REGION Network 32: data management MV01
   RUNG wire#powerrail
      Contact( "EM_OK" )
      wire#w1
      I_Contact( "MV01_Close" )
      wire#w2
      Coil( "fill_unit1".CONTROL_SIGNALS.SW_GATE0 )
   END_RUNG
   RUNG wire#w2
      { S7_Templates := "SrcType := DInt"; S7_GenerateENO := "TRUE" } Add(in1 := "Memory encoder".Encoder_CH00, in2 := "fill_unit1".ACT_CNTV0, out => #CNT_Act_0)
      { S7_Templates := "SrcType := DInt"; S7_GenerateENO := "TRUE" } Div(in1 := #CNT_Act_0, in2 := 100, out => #CNTV0_100)
      { S7_GenerateENO := "TRUE" } Move(in := #CNTV0_100, out1 => "Memory encoder".Encoder_CH00_10)
   END_RUNG
   RUNG wire#w1
      I_Contact( "fill_unit1".CONTROL_SIGNALS.SW_GATE0 )
      wire#w3
      { S7_GenerateENO := "TRUE" } Move(in := 0, out1 => "Memory encoder".Encoder_CH00_10)
   END_RUNG
   RUNG wire#w3
      { S7_GenerateENO := "TRUE" } Move(in := INT#0, out1 => "Memory encoder".Encoder_CH00)
   END_RUNG
   RUNG wire#w1
      "Signal linearization"(IN0 := "ON", Analog_input := "Memory encoder".Encoder_CH00_10, Coeff := "Coeff".COEFF_TRASM_MV01, Zero := "Coeff".ZERO_TRASM_MV01, OutValue => "Data".Pot_MV01, Out_of_range => "Allarm".Pot_MV01_OFR)
   END_RUNG
   // the same network as SCL:
   // ENO of a box is taken as its EN; it also drops when the box reports an error
   "fill_unit1".CONTROL_SIGNALS.SW_GATE0 := "EM_OK" AND NOT "MV01_Close";
   IF "fill_unit1".CONTROL_SIGNALS.SW_GATE0 THEN
       #CNT_Act_0 := "Memory encoder".Encoder_CH00 + "fill_unit1".ACT_CNTV0;
       #CNTV0_100 := #CNT_Act_0 / 100;
       "Memory encoder".Encoder_CH00_10 := #CNTV0_100;
   END_IF;
   IF "EM_OK" AND NOT "fill_unit1".CONTROL_SIGNALS.SW_GATE0 THEN
       "Memory encoder".Encoder_CH00_10 := 0;
       "Memory encoder".Encoder_CH00 := INT#0;
   END_IF;
   IF "EM_OK" THEN
       "Signal linearization"(IN0 := "ON",
                              Analog_input := "Memory encoder".Encoder_CH00_10,
                              Coeff := "Coeff".COEFF_TRASM_MV01,
                              Zero := "Coeff".ZERO_TRASM_MV01,
                              OutValue => "Data".Pot_MV01,
                              Out_of_range => "Allarm".Pot_MV01_OFR);
   END_IF;
END_REGION

REGION Network 33: data management MV02
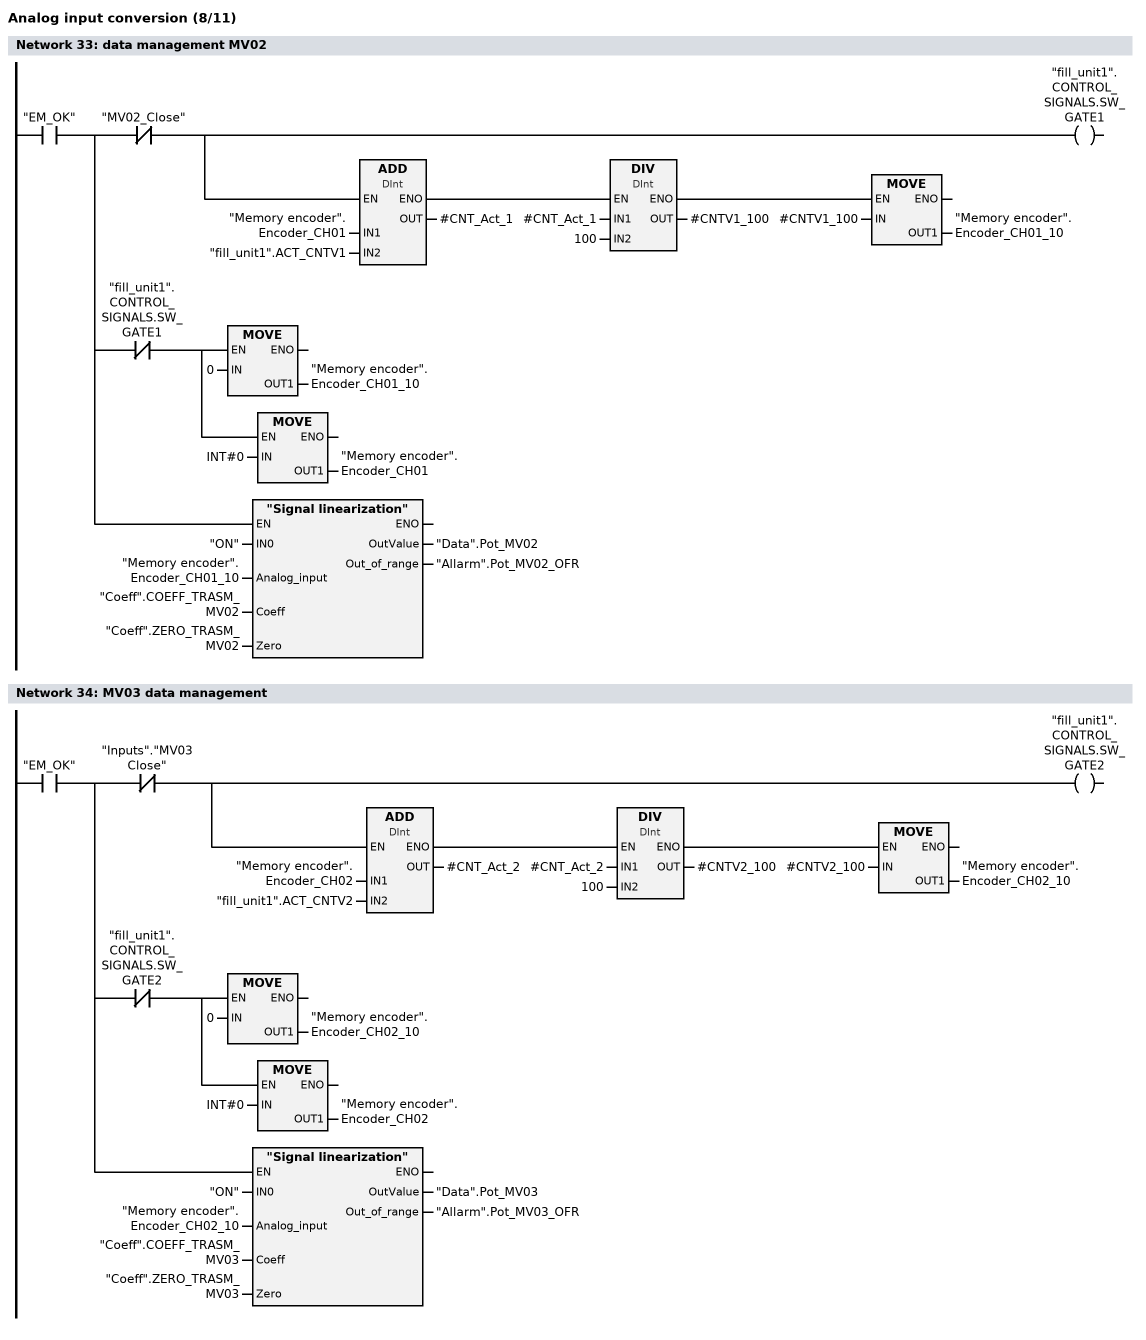
   RUNG wire#powerrail
      Contact( "EM_OK" )
      wire#w1
      I_Contact( "MV02_Close" )
      wire#w2
      Coil( "fill_unit1".CONTROL_SIGNALS.SW_GATE1 )
   END_RUNG
   RUNG wire#w2
      { S7_Templates := "SrcType := DInt"; S7_GenerateENO := "TRUE" } Add(in1 := "Memory encoder".Encoder_CH01, in2 := "fill_unit1".ACT_CNTV1, out => #CNT_Act_1)
      { S7_Templates := "SrcType := DInt"; S7_GenerateENO := "TRUE" } Div(in1 := #CNT_Act_1, in2 := 100, out => #CNTV1_100)
      { S7_GenerateENO := "TRUE" } Move(in := #CNTV1_100, out1 => "Memory encoder".Encoder_CH01_10)
   END_RUNG
   RUNG wire#w1
      I_Contact( "fill_unit1".CONTROL_SIGNALS.SW_GATE1 )
      wire#w3
      { S7_GenerateENO := "TRUE" } Move(in := 0, out1 => "Memory encoder".Encoder_CH01_10)
   END_RUNG
   RUNG wire#w3
      { S7_GenerateENO := "TRUE" } Move(in := INT#0, out1 => "Memory encoder".Encoder_CH01)
   END_RUNG
   RUNG wire#w1
      "Signal linearization"(IN0 := "ON", Analog_input := "Memory encoder".Encoder_CH01_10, Coeff := "Coeff".COEFF_TRASM_MV02, Zero := "Coeff".ZERO_TRASM_MV02, OutValue => "Data".Pot_MV02, Out_of_range => "Allarm".Pot_MV02_OFR)
   END_RUNG
   // the same network as SCL:
   // ENO of a box is taken as its EN; it also drops when the box reports an error
   "fill_unit1".CONTROL_SIGNALS.SW_GATE1 := "EM_OK" AND NOT "MV02_Close";
   IF "fill_unit1".CONTROL_SIGNALS.SW_GATE1 THEN
       #CNT_Act_1 := "Memory encoder".Encoder_CH01 + "fill_unit1".ACT_CNTV1;
       #CNTV1_100 := #CNT_Act_1 / 100;
       "Memory encoder".Encoder_CH01_10 := #CNTV1_100;
   END_IF;
   IF "EM_OK" AND NOT "fill_unit1".CONTROL_SIGNALS.SW_GATE1 THEN
       "Memory encoder".Encoder_CH01_10 := 0;
       "Memory encoder".Encoder_CH01 := INT#0;
   END_IF;
   IF "EM_OK" THEN
       "Signal linearization"(IN0 := "ON",
                              Analog_input := "Memory encoder".Encoder_CH01_10,
                              Coeff := "Coeff".COEFF_TRASM_MV02,
                              Zero := "Coeff".ZERO_TRASM_MV02,
                              OutValue => "Data".Pot_MV02,
                              Out_of_range => "Allarm".Pot_MV02_OFR);
   END_IF;
END_REGION

REGION Network 34: MV03 data management
   RUNG wire#powerrail
      Contact( "EM_OK" )
      wire#w1
      I_Contact( "Inputs"."MV03 Close" )
      wire#w2
      Coil( "fill_unit1".CONTROL_SIGNALS.SW_GATE2 )
   END_RUNG
   RUNG wire#w2
      { S7_Templates := "SrcType := DInt"; S7_GenerateENO := "TRUE" } Add(in1 := "Memory encoder".Encoder_CH02, in2 := "fill_unit1".ACT_CNTV2, out => #CNT_Act_2)
      { S7_Templates := "SrcType := DInt"; S7_GenerateENO := "TRUE" } Div(in1 := #CNT_Act_2, in2 := 100, out => #CNTV2_100)
      { S7_GenerateENO := "TRUE" } Move(in := #CNTV2_100, out1 => "Memory encoder".Encoder_CH02_10)
   END_RUNG
   RUNG wire#w1
      I_Contact( "fill_unit1".CONTROL_SIGNALS.SW_GATE2 )
      wire#w3
      { S7_GenerateENO := "TRUE" } Move(in := 0, out1 => "Memory encoder".Encoder_CH02_10)
   END_RUNG
   RUNG wire#w3
      { S7_GenerateENO := "TRUE" } Move(in := INT#0, out1 => "Memory encoder".Encoder_CH02)
   END_RUNG
   RUNG wire#w1
      "Signal linearization"(IN0 := "ON", Analog_input := "Memory encoder".Encoder_CH02_10, Coeff := "Coeff".COEFF_TRASM_MV03, Zero := "Coeff".ZERO_TRASM_MV03, OutValue => "Data".Pot_MV03, Out_of_range => "Allarm".Pot_MV03_OFR)
   END_RUNG
   // the same network as SCL:
   // ENO of a box is taken as its EN; it also drops when the box reports an error
   "fill_unit1".CONTROL_SIGNALS.SW_GATE2 := "EM_OK" AND NOT "Inputs"."MV03 Close";
   IF "fill_unit1".CONTROL_SIGNALS.SW_GATE2 THEN
       #CNT_Act_2 := "Memory encoder".Encoder_CH02 + "fill_unit1".ACT_CNTV2;
       #CNTV2_100 := #CNT_Act_2 / 100;
       "Memory encoder".Encoder_CH02_10 := #CNTV2_100;
   END_IF;
   IF "EM_OK" AND NOT "fill_unit1".CONTROL_SIGNALS.SW_GATE2 THEN
       "Memory encoder".Encoder_CH02_10 := 0;
       "Memory encoder".Encoder_CH02 := INT#0;
   END_IF;
   IF "EM_OK" THEN
       "Signal linearization"(IN0 := "ON",
                              Analog_input := "Memory encoder".Encoder_CH02_10,
                              Coeff := "Coeff".COEFF_TRASM_MV03,
                              Zero := "Coeff".ZERO_TRASM_MV03,
                              OutValue => "Data".Pot_MV03,
                              Out_of_range => "Allarm".Pot_MV03_OFR);
   END_IF;
END_REGION

REGION Network 35: MV05 data management
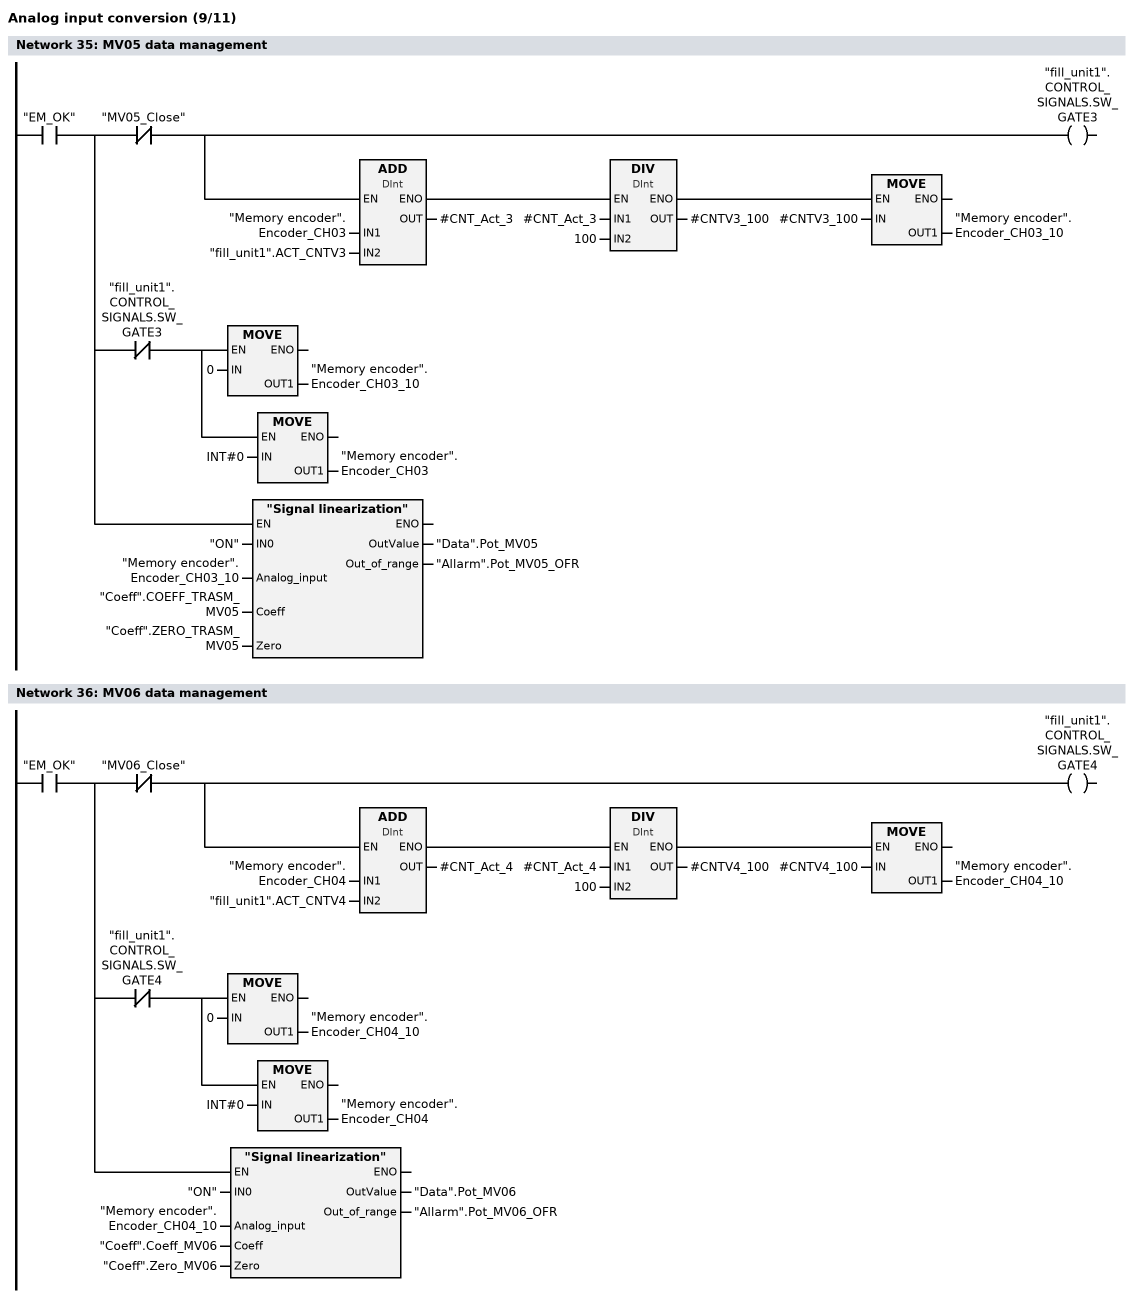
   RUNG wire#powerrail
      Contact( "EM_OK" )
      wire#w1
      I_Contact( "MV05_Close" )
      wire#w2
      Coil( "fill_unit1".CONTROL_SIGNALS.SW_GATE3 )
   END_RUNG
   RUNG wire#w2
      { S7_Templates := "SrcType := DInt"; S7_GenerateENO := "TRUE" } Add(in1 := "Memory encoder".Encoder_CH03, in2 := "fill_unit1".ACT_CNTV3, out => #CNT_Act_3)
      { S7_Templates := "SrcType := DInt"; S7_GenerateENO := "TRUE" } Div(in1 := #CNT_Act_3, in2 := 100, out => #CNTV3_100)
      { S7_GenerateENO := "TRUE" } Move(in := #CNTV3_100, out1 => "Memory encoder".Encoder_CH03_10)
   END_RUNG
   RUNG wire#w1
      I_Contact( "fill_unit1".CONTROL_SIGNALS.SW_GATE3 )
      wire#w3
      { S7_GenerateENO := "TRUE" } Move(in := 0, out1 => "Memory encoder".Encoder_CH03_10)
   END_RUNG
   RUNG wire#w3
      { S7_GenerateENO := "TRUE" } Move(in := INT#0, out1 => "Memory encoder".Encoder_CH03)
   END_RUNG
   RUNG wire#w1
      "Signal linearization"(IN0 := "ON", Analog_input := "Memory encoder".Encoder_CH03_10, Coeff := "Coeff".COEFF_TRASM_MV05, Zero := "Coeff".ZERO_TRASM_MV05, OutValue => "Data".Pot_MV05, Out_of_range => "Allarm".Pot_MV05_OFR)
   END_RUNG
   // the same network as SCL:
   // ENO of a box is taken as its EN; it also drops when the box reports an error
   "fill_unit1".CONTROL_SIGNALS.SW_GATE3 := "EM_OK" AND NOT "MV05_Close";
   IF "fill_unit1".CONTROL_SIGNALS.SW_GATE3 THEN
       #CNT_Act_3 := "Memory encoder".Encoder_CH03 + "fill_unit1".ACT_CNTV3;
       #CNTV3_100 := #CNT_Act_3 / 100;
       "Memory encoder".Encoder_CH03_10 := #CNTV3_100;
   END_IF;
   IF "EM_OK" AND NOT "fill_unit1".CONTROL_SIGNALS.SW_GATE3 THEN
       "Memory encoder".Encoder_CH03_10 := 0;
       "Memory encoder".Encoder_CH03 := INT#0;
   END_IF;
   IF "EM_OK" THEN
       "Signal linearization"(IN0 := "ON",
                              Analog_input := "Memory encoder".Encoder_CH03_10,
                              Coeff := "Coeff".COEFF_TRASM_MV05,
                              Zero := "Coeff".ZERO_TRASM_MV05,
                              OutValue => "Data".Pot_MV05,
                              Out_of_range => "Allarm".Pot_MV05_OFR);
   END_IF;
END_REGION

REGION Network 36: MV06 data management
   RUNG wire#powerrail
      Contact( "EM_OK" )
      wire#w1
      I_Contact( "MV06_Close" )
      wire#w2
      Coil( "fill_unit1".CONTROL_SIGNALS.SW_GATE4 )
   END_RUNG
   RUNG wire#w2
      { S7_Templates := "SrcType := DInt"; S7_GenerateENO := "TRUE" } Add(in1 := "Memory encoder".Encoder_CH04, in2 := "fill_unit1".ACT_CNTV4, out => #CNT_Act_4)
      { S7_Templates := "SrcType := DInt"; S7_GenerateENO := "TRUE" } Div(in1 := #CNT_Act_4, in2 := 100, out => #CNTV4_100)
      { S7_GenerateENO := "TRUE" } Move(in := #CNTV4_100, out1 => "Memory encoder".Encoder_CH04_10)
   END_RUNG
   RUNG wire#w1
      I_Contact( "fill_unit1".CONTROL_SIGNALS.SW_GATE4 )
      wire#w3
      { S7_GenerateENO := "TRUE" } Move(in := 0, out1 => "Memory encoder".Encoder_CH04_10)
   END_RUNG
   RUNG wire#w3
      { S7_GenerateENO := "TRUE" } Move(in := INT#0, out1 => "Memory encoder".Encoder_CH04)
   END_RUNG
   RUNG wire#w1
      "Signal linearization"(IN0 := "ON", Analog_input := "Memory encoder".Encoder_CH04_10, Coeff := "Coeff".Coeff_MV06, Zero := "Coeff".Zero_MV06, OutValue => "Data".Pot_MV06, Out_of_range => "Allarm".Pot_MV06_OFR)
   END_RUNG
   // the same network as SCL:
   // ENO of a box is taken as its EN; it also drops when the box reports an error
   "fill_unit1".CONTROL_SIGNALS.SW_GATE4 := "EM_OK" AND NOT "MV06_Close";
   IF "fill_unit1".CONTROL_SIGNALS.SW_GATE4 THEN
       #CNT_Act_4 := "Memory encoder".Encoder_CH04 + "fill_unit1".ACT_CNTV4;
       #CNTV4_100 := #CNT_Act_4 / 100;
       "Memory encoder".Encoder_CH04_10 := #CNTV4_100;
   END_IF;
   IF "EM_OK" AND NOT "fill_unit1".CONTROL_SIGNALS.SW_GATE4 THEN
       "Memory encoder".Encoder_CH04_10 := 0;
       "Memory encoder".Encoder_CH04 := INT#0;
   END_IF;
   IF "EM_OK" THEN
       "Signal linearization"(IN0 := "ON",
                              Analog_input := "Memory encoder".Encoder_CH04_10,
                              Coeff := "Coeff".Coeff_MV06,
                              Zero := "Coeff".Zero_MV06,
                              OutValue => "Data".Pot_MV06,
                              Out_of_range => "Allarm".Pot_MV06_OFR);
   END_IF;
END_REGION

REGION Network 37: FN-02 FAN
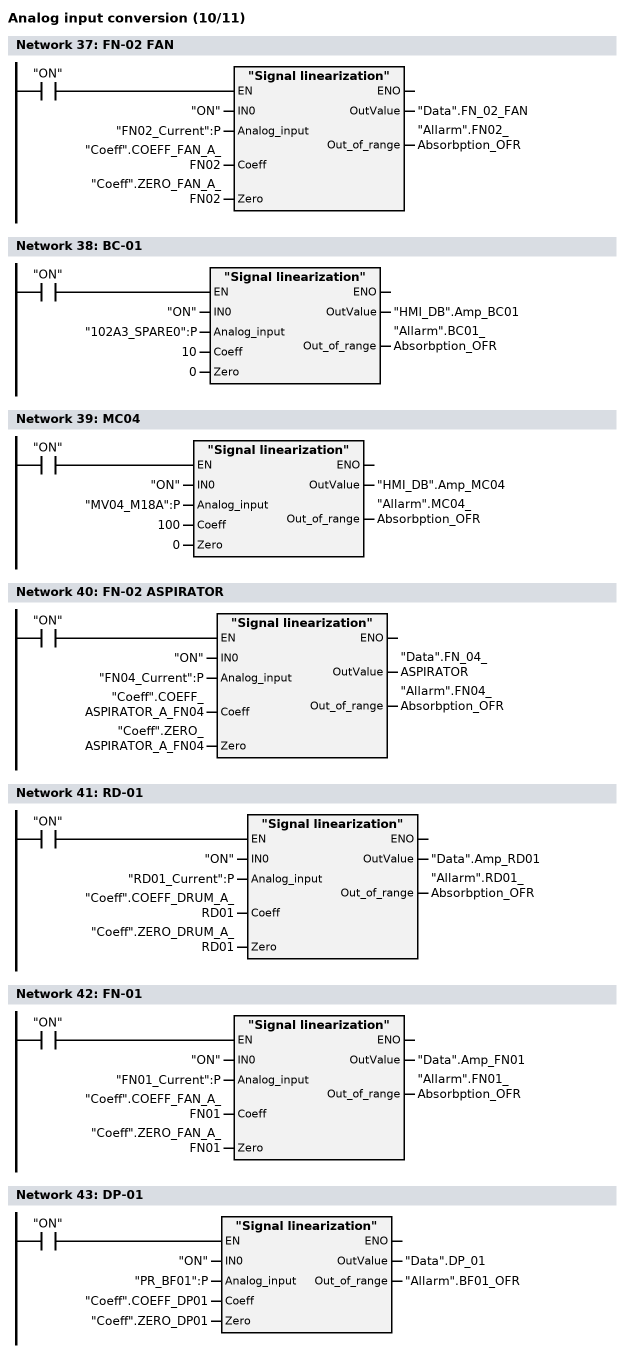
   RUNG wire#powerrail
      Contact( "ON" )
      "Signal linearization"(IN0 := "ON", Analog_input := "FN02_Current":P, Coeff := "Coeff".COEFF_FAN_A_FN02, Zero := "Coeff".ZERO_FAN_A_FN02, OutValue => "Data".FN_02_FAN, Out_of_range => "Allarm".FN02_Absorbption_OFR)
   END_RUNG
   // the same network as SCL:
   IF "ON" THEN
       "Signal linearization"(IN0 := "ON",
                              Analog_input := "FN02_Current":P,
                              Coeff := "Coeff".COEFF_FAN_A_FN02,
                              Zero := "Coeff".ZERO_FAN_A_FN02,
                              OutValue => "Data".FN_02_FAN,
                              Out_of_range => "Allarm".FN02_Absorbption_OFR);
   END_IF;
END_REGION

REGION Network 38: BC-01
   RUNG wire#powerrail
      Contact( "ON" )
      "Signal linearization"(IN0 := "ON", Analog_input := "102A3_SPARE0":P, Coeff := 10, Zero := 0, OutValue => "HMI_DB".Amp_BC01, Out_of_range => "Allarm".BC01_Absorbption_OFR)
   END_RUNG
   // the same network as SCL:
   IF "ON" THEN
       "Signal linearization"(IN0 := "ON",
                              Analog_input := "102A3_SPARE0":P,
                              Coeff := 10,
                              Zero := 0,
                              OutValue => "HMI_DB".Amp_BC01,
                              Out_of_range => "Allarm".BC01_Absorbption_OFR);
   END_IF;
END_REGION

REGION Network 39: MC04
   RUNG wire#powerrail
      Contact( "ON" )
      "Signal linearization"(IN0 := "ON", Analog_input := "MV04_M18A":P, Coeff := 100, Zero := 0, OutValue => "HMI_DB".Amp_MC04, Out_of_range => "Allarm".MC04_Absorbption_OFR)
   END_RUNG
   // the same network as SCL:
   IF "ON" THEN
       "Signal linearization"(IN0 := "ON",
                              Analog_input := "MV04_M18A":P,
                              Coeff := 100,
                              Zero := 0,
                              OutValue => "HMI_DB".Amp_MC04,
                              Out_of_range => "Allarm".MC04_Absorbption_OFR);
   END_IF;
END_REGION

REGION Network 40: FN-02 ASPIRATOR
   RUNG wire#powerrail
      Contact( "ON" )
      "Signal linearization"(IN0 := "ON", Analog_input := "FN04_Current":P, Coeff := "Coeff".COEFF_ASPIRATOR_A_FN04, Zero := "Coeff".ZERO_ASPIRATOR_A_FN04, OutValue => "Data".FN_04_ASPIRATOR, Out_of_range => "Allarm".FN04_Absorbption_OFR)
   END_RUNG
   // the same network as SCL:
   IF "ON" THEN
       "Signal linearization"(IN0 := "ON",
                              Analog_input := "FN04_Current":P,
                              Coeff := "Coeff".COEFF_ASPIRATOR_A_FN04,
                              Zero := "Coeff".ZERO_ASPIRATOR_A_FN04,
                              OutValue => "Data".FN_04_ASPIRATOR,
                              Out_of_range => "Allarm".FN04_Absorbption_OFR);
   END_IF;
END_REGION

REGION Network 41: RD-01
   RUNG wire#powerrail
      Contact( "ON" )
      "Signal linearization"(IN0 := "ON", Analog_input := "RD01_Current":P, Coeff := "Coeff".COEFF_DRUM_A_RD01, Zero := "Coeff".ZERO_DRUM_A_RD01, OutValue => "Data".Amp_RD01, Out_of_range => "Allarm".RD01_Absorbption_OFR)
   END_RUNG
   // the same network as SCL:
   IF "ON" THEN
       "Signal linearization"(IN0 := "ON",
                              Analog_input := "RD01_Current":P,
                              Coeff := "Coeff".COEFF_DRUM_A_RD01,
                              Zero := "Coeff".ZERO_DRUM_A_RD01,
                              OutValue => "Data".Amp_RD01,
                              Out_of_range => "Allarm".RD01_Absorbption_OFR);
   END_IF;
END_REGION

REGION Network 42: FN-01
   RUNG wire#powerrail
      Contact( "ON" )
      "Signal linearization"(IN0 := "ON", Analog_input := "FN01_Current":P, Coeff := "Coeff".COEFF_FAN_A_FN01, Zero := "Coeff".ZERO_FAN_A_FN01, OutValue => "Data".Amp_FN01, Out_of_range => "Allarm".FN01_Absorbption_OFR)
   END_RUNG
   // the same network as SCL:
   IF "ON" THEN
       "Signal linearization"(IN0 := "ON",
                              Analog_input := "FN01_Current":P,
                              Coeff := "Coeff".COEFF_FAN_A_FN01,
                              Zero := "Coeff".ZERO_FAN_A_FN01,
                              OutValue => "Data".Amp_FN01,
                              Out_of_range => "Allarm".FN01_Absorbption_OFR);
   END_IF;
END_REGION

REGION Network 43: DP-01
   RUNG wire#powerrail
      Contact( "ON" )
      "Signal linearization"(IN0 := "ON", Analog_input := "PR_BF01":P, Coeff := "Coeff".COEFF_DP01, Zero := "Coeff".ZERO_DP01, OutValue => "Data".DP_01, Out_of_range => "Allarm".BF01_OFR)
   END_RUNG
   // the same network as SCL:
   IF "ON" THEN
       "Signal linearization"(IN0 := "ON",
                              Analog_input := "PR_BF01":P,
                              Coeff := "Coeff".COEFF_DP01,
                              Zero := "Coeff".ZERO_DP01,
                              OutValue => "Data".DP_01,
                              Out_of_range => "Allarm".BF01_OFR);
   END_IF;
END_REGION

REGION Network 44: DP-02
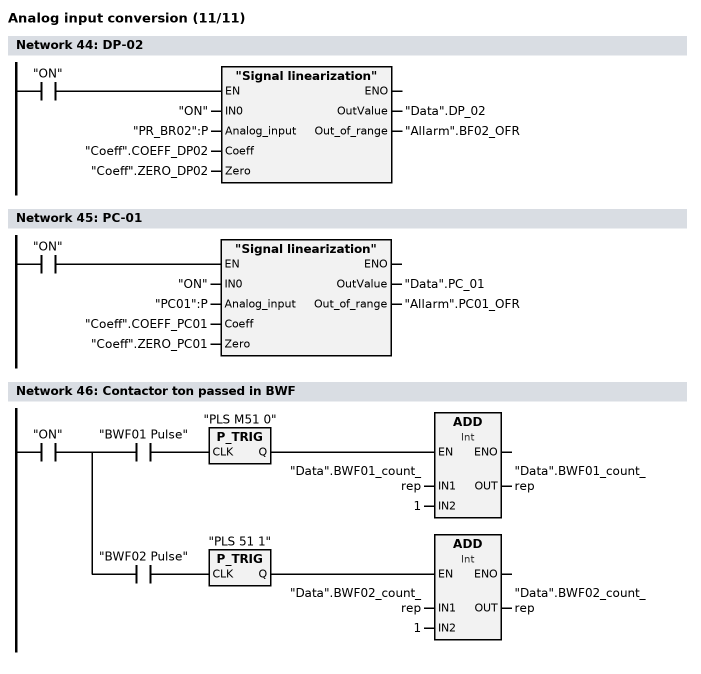
   RUNG wire#powerrail
      Contact( "ON" )
      "Signal linearization"(IN0 := "ON", Analog_input := "PR_BR02":P, Coeff := "Coeff".COEFF_DP02, Zero := "Coeff".ZERO_DP02, OutValue => "Data".DP_02, Out_of_range => "Allarm".BF02_OFR)
   END_RUNG
   // the same network as SCL:
   IF "ON" THEN
       "Signal linearization"(IN0 := "ON",
                              Analog_input := "PR_BR02":P,
                              Coeff := "Coeff".COEFF_DP02,
                              Zero := "Coeff".ZERO_DP02,
                              OutValue => "Data".DP_02,
                              Out_of_range => "Allarm".BF02_OFR);
   END_IF;
END_REGION

REGION Network 45: PC-01
   RUNG wire#powerrail
      Contact( "ON" )
      "Signal linearization"(IN0 := "ON", Analog_input := "PC01":P, Coeff := "Coeff".COEFF_PC01, Zero := "Coeff".ZERO_PC01, OutValue => "Data".PC_01, Out_of_range => "Allarm".PC01_OFR)
   END_RUNG
   // the same network as SCL:
   IF "ON" THEN
       "Signal linearization"(IN0 := "ON",
                              Analog_input := "PC01":P,
                              Coeff := "Coeff".COEFF_PC01,
                              Zero := "Coeff".ZERO_PC01,
                              OutValue => "Data".PC_01,
                              Out_of_range => "Allarm".PC01_OFR);
   END_IF;
END_REGION

REGION Network 46: Contactor ton passed in BWF
   RUNG wire#powerrail
      Contact( "ON" )
      wire#w1
      Contact( "BWF01 Pulse" )
      P_Trig( "PLS M51 0" )
      { S7_Templates := "SrcType := Int"; S7_GenerateENO := "TRUE" } Add(in1 := "Data".BWF01_count_rep, in2 := 1, out => "Data".BWF01_count_rep)
   END_RUNG
   RUNG wire#w1
      Contact( "BWF02 Pulse" )
      P_Trig( "PLS 51 1" )
      { S7_Templates := "SrcType := Int"; S7_GenerateENO := "TRUE" } Add(in1 := "Data".BWF02_count_rep, in2 := 1, out => "Data".BWF02_count_rep)
   END_RUNG
   // the same network as SCL:
   #_w1 := "ON" AND "BWF01 Pulse";
   #_w2 := #_w1 AND NOT "PLS M51 0";   // rising edge
   "PLS M51 0" := #_w1;
   IF #_w2 THEN "Data".BWF01_count_rep := "Data".BWF01_count_rep + 1; END_IF;
   #_w3 := "ON" AND "BWF02 Pulse";
   #_w4 := #_w3 AND NOT "PLS 51 1";   // rising edge
   "PLS 51 1" := #_w3;
   IF #_w4 THEN "Data".BWF02_count_rep := "Data".BWF02_count_rep + 1; END_IF;
END_REGION
END_FUNCTION

FUNCTION "Allarms 1" : Void   // FC4, LAD
TITLE = Motors alarms
{ S7_Optimized_Access := 'FALSE' }
VERSION : 0.1
   VAR_TEMP   // added for the SCL form of the ladder/FBD networks
      _w1 : Bool;
      _w2 : Bool;
      _w3 : Bool;
      _w4 : Bool;
      _w5 : Bool;
   END_VAR
BEGIN

REGION Network 1: BWF01
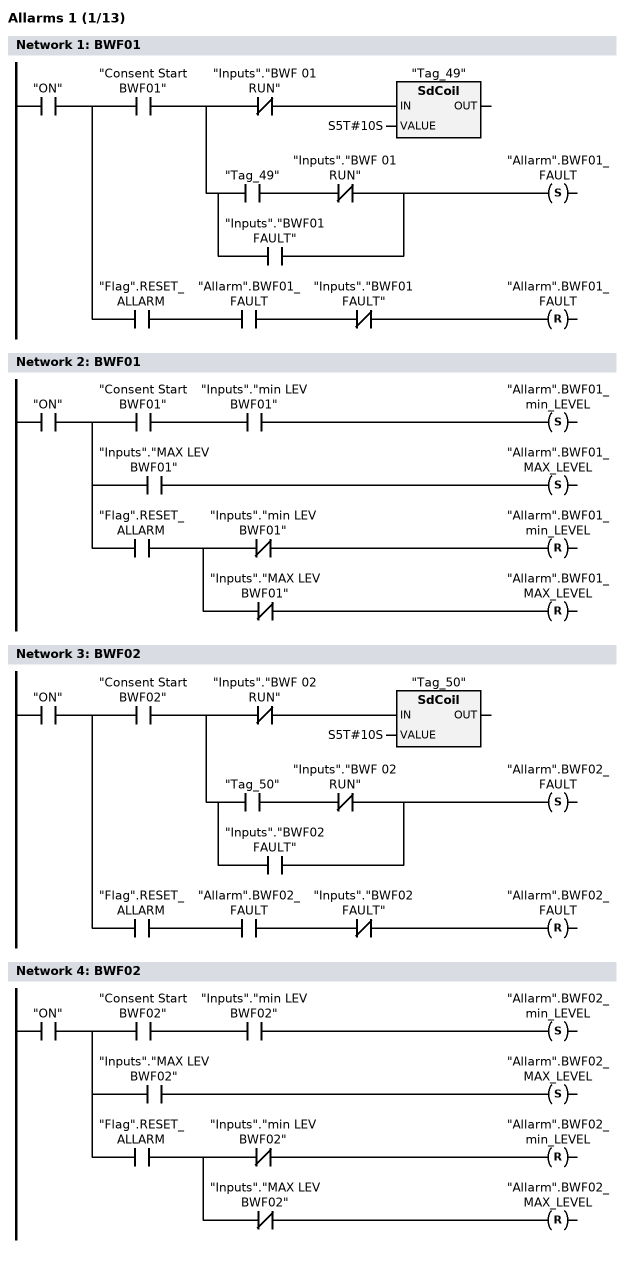
   // no SCL statement known for SdCoil: written as a call
   #_w1 := "ON" AND "Consent Start BWF01";
   #_w2 := "ON";
   SdCoil(in := #_w1 AND NOT "Inputs"."BWF 01 RUN", value := S5T#10S, operand := "Tag_49");
   IF #_w1 AND (("Tag_49" AND NOT "Inputs"."BWF 01 RUN") OR "Inputs"."BWF01 FAULT") THEN
       "Allarm".BWF01_FAULT := TRUE;
   END_IF;
   IF #_w2 AND "Flag".RESET_ALLARM AND "Allarm".BWF01_FAULT AND NOT "Inputs"."BWF01 FAULT" THEN
       "Allarm".BWF01_FAULT := FALSE;
   END_IF;
END_REGION

REGION Network 2: BWF01
   RUNG wire#powerrail
      Contact( "ON" )
      wire#w1
      Contact( "Consent Start BWF01" )
      Contact( "Inputs"."min LEV BWF01" )
      S_Coil( "Allarm".BWF01_min_LEVEL )
   END_RUNG
   RUNG wire#w1
      Contact( "Inputs"."MAX LEV BWF01" )
      S_Coil( "Allarm".BWF01_MAX_LEVEL )
   END_RUNG
   RUNG wire#w1
      Contact( "Flag".RESET_ALLARM )
      wire#w2
      I_Contact( "Inputs"."min LEV BWF01" )
      R_Coil( "Allarm".BWF01_min_LEVEL )
   END_RUNG
   RUNG wire#w2
      I_Contact( "Inputs"."MAX LEV BWF01" )
      R_Coil( "Allarm".BWF01_MAX_LEVEL )
   END_RUNG
   // the same network as SCL:
   IF "ON" AND "Consent Start BWF01" AND "Inputs"."min LEV BWF01" THEN
       "Allarm".BWF01_min_LEVEL := TRUE;
   END_IF;
   IF "ON" AND "Inputs"."MAX LEV BWF01" THEN "Allarm".BWF01_MAX_LEVEL := TRUE; END_IF;
   #_w1 := "ON" AND "Flag".RESET_ALLARM;
   IF #_w1 AND NOT "Inputs"."min LEV BWF01" THEN "Allarm".BWF01_min_LEVEL := FALSE; END_IF;
   IF #_w1 AND NOT "Inputs"."MAX LEV BWF01" THEN "Allarm".BWF01_MAX_LEVEL := FALSE; END_IF;
END_REGION

REGION Network 3: BWF02
   // no SCL statement known for SdCoil: written as a call
   #_w1 := "ON" AND "Consent Start BWF02";
   #_w2 := "ON";
   SdCoil(in := #_w1 AND NOT "Inputs"."BWF 02 RUN", value := S5T#10S, operand := "Tag_50");
   IF #_w1 AND (("Tag_50" AND NOT "Inputs"."BWF 02 RUN") OR "Inputs"."BWF02 FAULT") THEN
       "Allarm".BWF02_FAULT := TRUE;
   END_IF;
   IF #_w2 AND "Flag".RESET_ALLARM AND "Allarm".BWF02_FAULT AND NOT "Inputs"."BWF02 FAULT" THEN
       "Allarm".BWF02_FAULT := FALSE;
   END_IF;
END_REGION

REGION Network 4: BWF02
   RUNG wire#powerrail
      Contact( "ON" )
      wire#w1
      Contact( "Consent Start BWF02" )
      Contact( "Inputs"."min LEV BWF02" )
      S_Coil( "Allarm".BWF02_min_LEVEL )
   END_RUNG
   RUNG wire#w1
      Contact( "Inputs"."MAX LEV BWF02" )
      S_Coil( "Allarm".BWF02_MAX_LEVEL )
   END_RUNG
   RUNG wire#w1
      Contact( "Flag".RESET_ALLARM )
      wire#w2
      I_Contact( "Inputs"."min LEV BWF02" )
      R_Coil( "Allarm".BWF02_min_LEVEL )
   END_RUNG
   RUNG wire#w2
      I_Contact( "Inputs"."MAX LEV BWF02" )
      R_Coil( "Allarm".BWF02_MAX_LEVEL )
   END_RUNG
   // the same network as SCL:
   IF "ON" AND "Consent Start BWF02" AND "Inputs"."min LEV BWF02" THEN
       "Allarm".BWF02_min_LEVEL := TRUE;
   END_IF;
   IF "ON" AND "Inputs"."MAX LEV BWF02" THEN "Allarm".BWF02_MAX_LEVEL := TRUE; END_IF;
   #_w1 := "ON" AND "Flag".RESET_ALLARM;
   IF #_w1 AND NOT "Inputs"."min LEV BWF02" THEN "Allarm".BWF02_min_LEVEL := FALSE; END_IF;
   IF #_w1 AND NOT "Inputs"."MAX LEV BWF02" THEN "Allarm".BWF02_MAX_LEVEL := FALSE; END_IF;
END_REGION

REGION Network 5: BC01
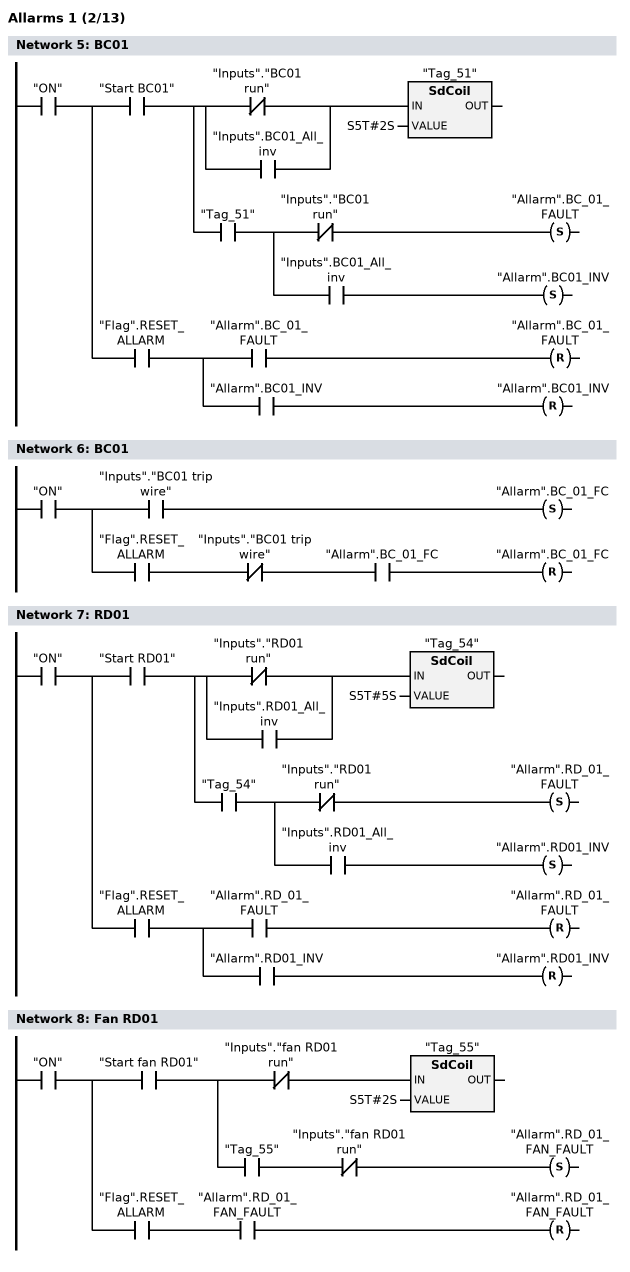
   // no SCL statement known for SdCoil: written as a call
   #_w1 := "ON" AND "Start BC01";
   #_w2 := "ON";
   SdCoil(in := #_w1 AND (NOT "Inputs"."BC01 run" OR "Inputs".BC01_All_inv),
          value := S5T#2S,
          operand := "Tag_51");
   #_w3 := #_w1 AND "Tag_51";
   IF #_w3 AND NOT "Inputs"."BC01 run" THEN "Allarm".BC_01_FAULT := TRUE; END_IF;
   IF #_w3 AND "Inputs".BC01_All_inv THEN "Allarm".BC01_INV := TRUE; END_IF;
   #_w4 := #_w2 AND "Flag".RESET_ALLARM;
   IF #_w4 AND "Allarm".BC_01_FAULT THEN "Allarm".BC_01_FAULT := FALSE; END_IF;
   IF #_w4 AND "Allarm".BC01_INV THEN "Allarm".BC01_INV := FALSE; END_IF;
END_REGION

REGION Network 6: BC01
   RUNG wire#powerrail
      Contact( "ON" )
      wire#w1
      Contact( "Inputs"."BC01 trip wire" )
      S_Coil( "Allarm".BC_01_FC )
   END_RUNG
   RUNG wire#w1
      Contact( "Flag".RESET_ALLARM )
      I_Contact( "Inputs"."BC01 trip wire" )
      Contact( "Allarm".BC_01_FC )
      R_Coil( "Allarm".BC_01_FC )
   END_RUNG
   // the same network as SCL:
   IF "ON" AND "Inputs"."BC01 trip wire" THEN "Allarm".BC_01_FC := TRUE; END_IF;
   IF "ON" AND "Flag".RESET_ALLARM AND NOT "Inputs"."BC01 trip wire" AND "Allarm".BC_01_FC THEN
       "Allarm".BC_01_FC := FALSE;
   END_IF;
END_REGION

REGION Network 7: RD01
   // no SCL statement known for SdCoil: written as a call
   #_w1 := "ON" AND "Start RD01";
   #_w2 := "ON";
   SdCoil(in := #_w1 AND (NOT "Inputs"."RD01 run" OR "Inputs".RD01_All_inv),
          value := S5T#5S,
          operand := "Tag_54");
   #_w3 := #_w1 AND "Tag_54";
   IF #_w3 AND NOT "Inputs"."RD01 run" THEN "Allarm".RD_01_FAULT := TRUE; END_IF;
   IF #_w3 AND "Inputs".RD01_All_inv THEN "Allarm".RD01_INV := TRUE; END_IF;
   #_w4 := #_w2 AND "Flag".RESET_ALLARM;
   IF #_w4 AND "Allarm".RD_01_FAULT THEN "Allarm".RD_01_FAULT := FALSE; END_IF;
   IF #_w4 AND "Allarm".RD01_INV THEN "Allarm".RD01_INV := FALSE; END_IF;
END_REGION

REGION Network 8: Fan RD01
   // no SCL statement known for SdCoil: written as a call
   #_w1 := "ON" AND "Start fan RD01";
   #_w2 := "ON";
   SdCoil(in := #_w1 AND NOT "Inputs"."fan RD01 run", value := S5T#2S, operand := "Tag_55");
   IF #_w1 AND "Tag_55" AND NOT "Inputs"."fan RD01 run" THEN "Allarm".RD_01_FAN_FAULT := TRUE; END_IF;
   IF #_w2 AND "Flag".RESET_ALLARM AND "Allarm".RD_01_FAN_FAULT THEN
       "Allarm".RD_01_FAN_FAULT := FALSE;
   END_IF;
END_REGION

REGION Network 9: Spare motor
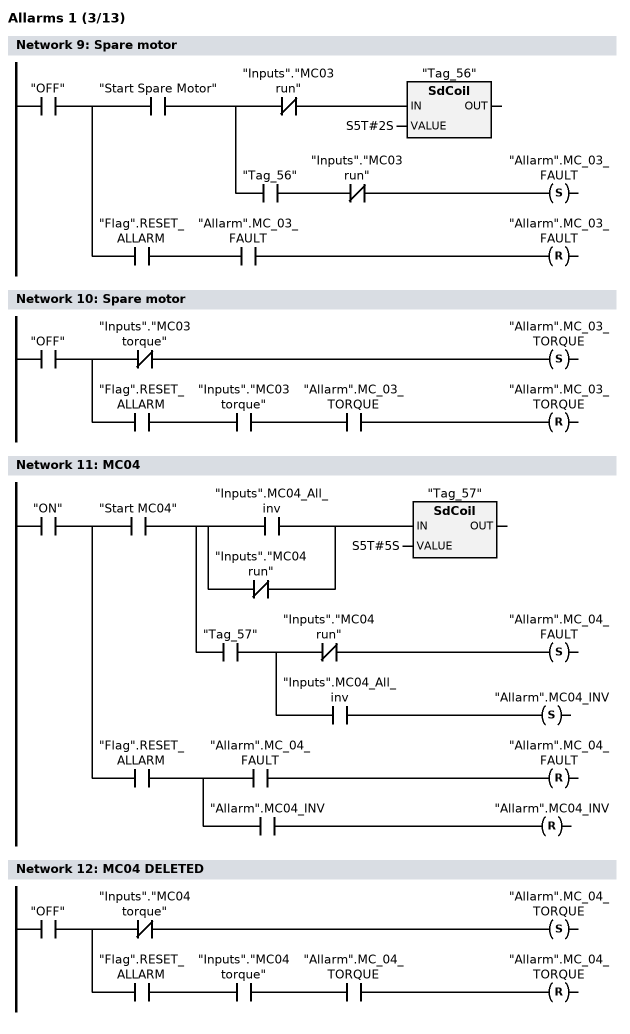
   // no SCL statement known for SdCoil: written as a call
   #_w1 := "OFF" AND "Start Spare Motor";
   #_w2 := "OFF";
   SdCoil(in := #_w1 AND NOT "Inputs"."MC03 run", value := S5T#2S, operand := "Tag_56");
   IF #_w1 AND "Tag_56" AND NOT "Inputs"."MC03 run" THEN "Allarm".MC_03_FAULT := TRUE; END_IF;
   IF #_w2 AND "Flag".RESET_ALLARM AND "Allarm".MC_03_FAULT THEN "Allarm".MC_03_FAULT := FALSE; END_IF;
END_REGION

REGION Network 10: Spare motor
   RUNG wire#powerrail
      Contact( "OFF" )
      wire#w1
      I_Contact( "Inputs"."MC03 torque" )
      S_Coil( "Allarm".MC_03_TORQUE )
   END_RUNG
   RUNG wire#w1
      Contact( "Flag".RESET_ALLARM )
      Contact( "Inputs"."MC03 torque" )
      Contact( "Allarm".MC_03_TORQUE )
      R_Coil( "Allarm".MC_03_TORQUE )
   END_RUNG
   // the same network as SCL:
   IF "OFF" AND NOT "Inputs"."MC03 torque" THEN "Allarm".MC_03_TORQUE := TRUE; END_IF;
   IF "OFF" AND "Flag".RESET_ALLARM AND "Inputs"."MC03 torque" AND "Allarm".MC_03_TORQUE THEN
       "Allarm".MC_03_TORQUE := FALSE;
   END_IF;
END_REGION

REGION Network 11: MC04
   // no SCL statement known for SdCoil: written as a call
   #_w1 := "ON" AND "Start MC04";
   #_w2 := "ON";
   SdCoil(in := #_w1 AND ("Inputs".MC04_All_inv OR NOT "Inputs"."MC04 run"),
          value := S5T#5S,
          operand := "Tag_57");
   #_w3 := #_w1 AND "Tag_57";
   IF #_w3 AND NOT "Inputs"."MC04 run" THEN "Allarm".MC_04_FAULT := TRUE; END_IF;
   IF #_w3 AND "Inputs".MC04_All_inv THEN "Allarm".MC04_INV := TRUE; END_IF;
   #_w4 := #_w2 AND "Flag".RESET_ALLARM;
   IF #_w4 AND "Allarm".MC_04_FAULT THEN "Allarm".MC_04_FAULT := FALSE; END_IF;
   IF #_w4 AND "Allarm".MC04_INV THEN "Allarm".MC04_INV := FALSE; END_IF;
END_REGION

REGION Network 12: MC04 DELETED
   RUNG wire#powerrail
      Contact( "OFF" )
      wire#w1
      I_Contact( "Inputs"."MC04 torque" )
      S_Coil( "Allarm".MC_04_TORQUE )
   END_RUNG
   RUNG wire#w1
      Contact( "Flag".RESET_ALLARM )
      Contact( "Inputs"."MC04 torque" )
      Contact( "Allarm".MC_04_TORQUE )
      R_Coil( "Allarm".MC_04_TORQUE )
   END_RUNG
   // the same network as SCL:
   IF "OFF" AND NOT "Inputs"."MC04 torque" THEN "Allarm".MC_04_TORQUE := TRUE; END_IF;
   IF "OFF" AND "Flag".RESET_ALLARM AND "Inputs"."MC04 torque" AND "Allarm".MC_04_TORQUE THEN
       "Allarm".MC_04_TORQUE := FALSE;
   END_IF;
END_REGION

REGION Network 13: MC05 DELETED
END_REGION

REGION Network 14: VS01
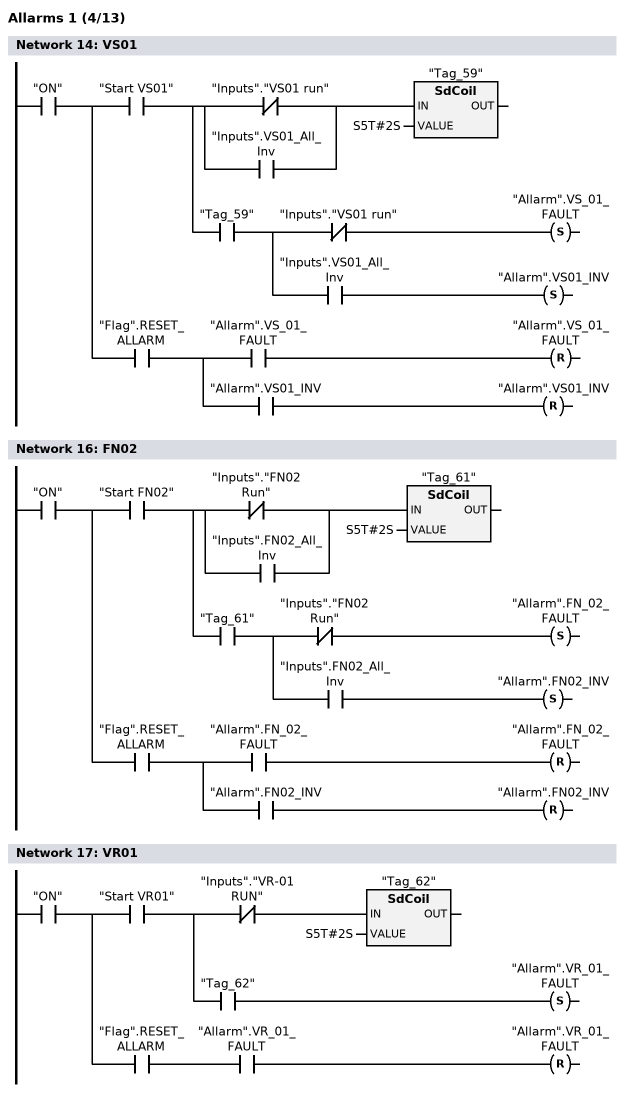
   // no SCL statement known for SdCoil: written as a call
   #_w1 := "ON" AND "Start VS01";
   #_w2 := "ON";
   SdCoil(in := #_w1 AND (NOT "Inputs"."VS01 run" OR "Inputs".VS01_All_Inv),
          value := S5T#2S,
          operand := "Tag_59");
   #_w3 := #_w1 AND "Tag_59";
   IF #_w3 AND NOT "Inputs"."VS01 run" THEN "Allarm".VS_01_FAULT := TRUE; END_IF;
   IF #_w3 AND "Inputs".VS01_All_Inv THEN "Allarm".VS01_INV := TRUE; END_IF;
   #_w4 := #_w2 AND "Flag".RESET_ALLARM;
   IF #_w4 AND "Allarm".VS_01_FAULT THEN "Allarm".VS_01_FAULT := FALSE; END_IF;
   IF #_w4 AND "Allarm".VS01_INV THEN "Allarm".VS01_INV := FALSE; END_IF;
END_REGION

REGION Network 15: SC12 DELETED
END_REGION

REGION Network 16: FN02
   // no SCL statement known for SdCoil: written as a call
   #_w1 := "ON" AND "Start FN02";
   #_w2 := "ON";
   SdCoil(in := #_w1 AND (NOT "Inputs"."FN02 Run" OR "Inputs".FN02_All_Inv),
          value := S5T#2S,
          operand := "Tag_61");
   #_w3 := #_w1 AND "Tag_61";
   IF #_w3 AND NOT "Inputs"."FN02 Run" THEN "Allarm".FN_02_FAULT := TRUE; END_IF;
   IF #_w3 AND "Inputs".FN02_All_Inv THEN "Allarm".FN02_INV := TRUE; END_IF;
   #_w4 := #_w2 AND "Flag".RESET_ALLARM;
   IF #_w4 AND "Allarm".FN_02_FAULT THEN "Allarm".FN_02_FAULT := FALSE; END_IF;
   IF #_w4 AND "Allarm".FN02_INV THEN "Allarm".FN02_INV := FALSE; END_IF;
END_REGION

REGION Network 17: VR01
   // no SCL statement known for SdCoil: written as a call
   #_w1 := "ON" AND "Start VR01";
   #_w2 := "ON";
   SdCoil(in := #_w1 AND NOT "Inputs"."VR-01 RUN", value := S5T#2S, operand := "Tag_62");
   IF #_w1 AND "Tag_62" THEN "Allarm".VR_01_FAULT := TRUE; END_IF;
   IF #_w2 AND "Flag".RESET_ALLARM AND "Allarm".VR_01_FAULT THEN "Allarm".VR_01_FAULT := FALSE; END_IF;
END_REGION

REGION Network 18: FN01
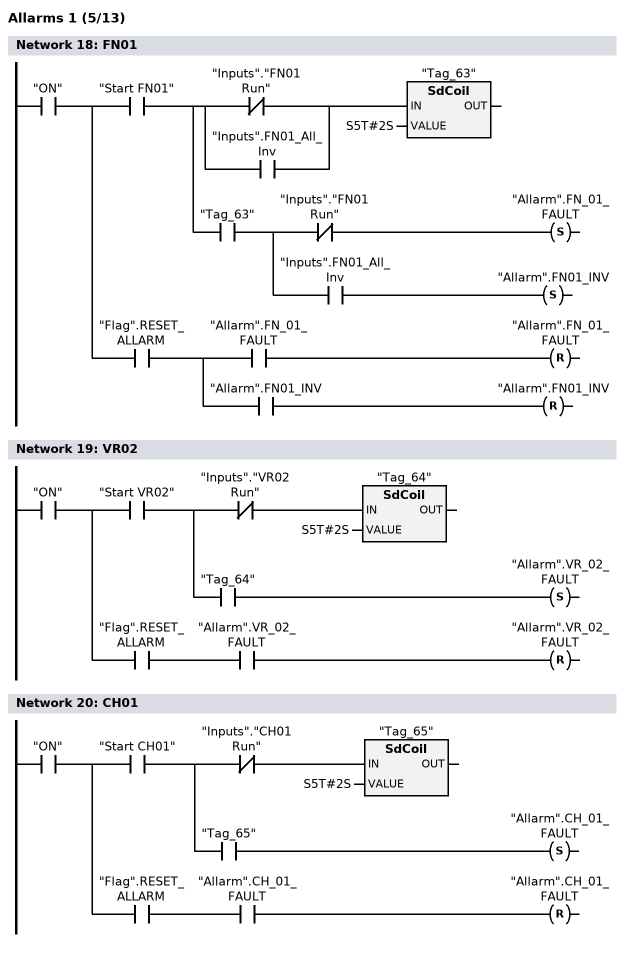
   // no SCL statement known for SdCoil: written as a call
   #_w1 := "ON" AND "Start FN01";
   #_w2 := "ON";
   SdCoil(in := #_w1 AND (NOT "Inputs"."FN01 Run" OR "Inputs".FN01_All_Inv),
          value := S5T#2S,
          operand := "Tag_63");
   #_w3 := #_w1 AND "Tag_63";
   IF #_w3 AND NOT "Inputs"."FN01 Run" THEN "Allarm".FN_01_FAULT := TRUE; END_IF;
   IF #_w3 AND "Inputs".FN01_All_Inv THEN "Allarm".FN01_INV := TRUE; END_IF;
   #_w4 := #_w2 AND "Flag".RESET_ALLARM;
   IF #_w4 AND "Allarm".FN_01_FAULT THEN "Allarm".FN_01_FAULT := FALSE; END_IF;
   IF #_w4 AND "Allarm".FN01_INV THEN "Allarm".FN01_INV := FALSE; END_IF;
END_REGION

REGION Network 19: VR02
   // no SCL statement known for SdCoil: written as a call
   #_w1 := "ON" AND "Start VR02";
   #_w2 := "ON";
   SdCoil(in := #_w1 AND NOT "Inputs"."VR02 Run", value := S5T#2S, operand := "Tag_64");
   IF #_w1 AND "Tag_64" THEN "Allarm".VR_02_FAULT := TRUE; END_IF;
   IF #_w2 AND "Flag".RESET_ALLARM AND "Allarm".VR_02_FAULT THEN "Allarm".VR_02_FAULT := FALSE; END_IF;
END_REGION

REGION Network 20: CH01
   // no SCL statement known for SdCoil: written as a call
   #_w1 := "ON" AND "Start CH01";
   #_w2 := "ON";
   SdCoil(in := #_w1 AND NOT "Inputs"."CH01 Run", value := S5T#2S, operand := "Tag_65");
   IF #_w1 AND "Tag_65" THEN "Allarm".CH_01_FAULT := TRUE; END_IF;
   IF #_w2 AND "Flag".RESET_ALLARM AND "Allarm".CH_01_FAULT THEN "Allarm".CH_01_FAULT := FALSE; END_IF;
END_REGION

REGION Network 21: FN03
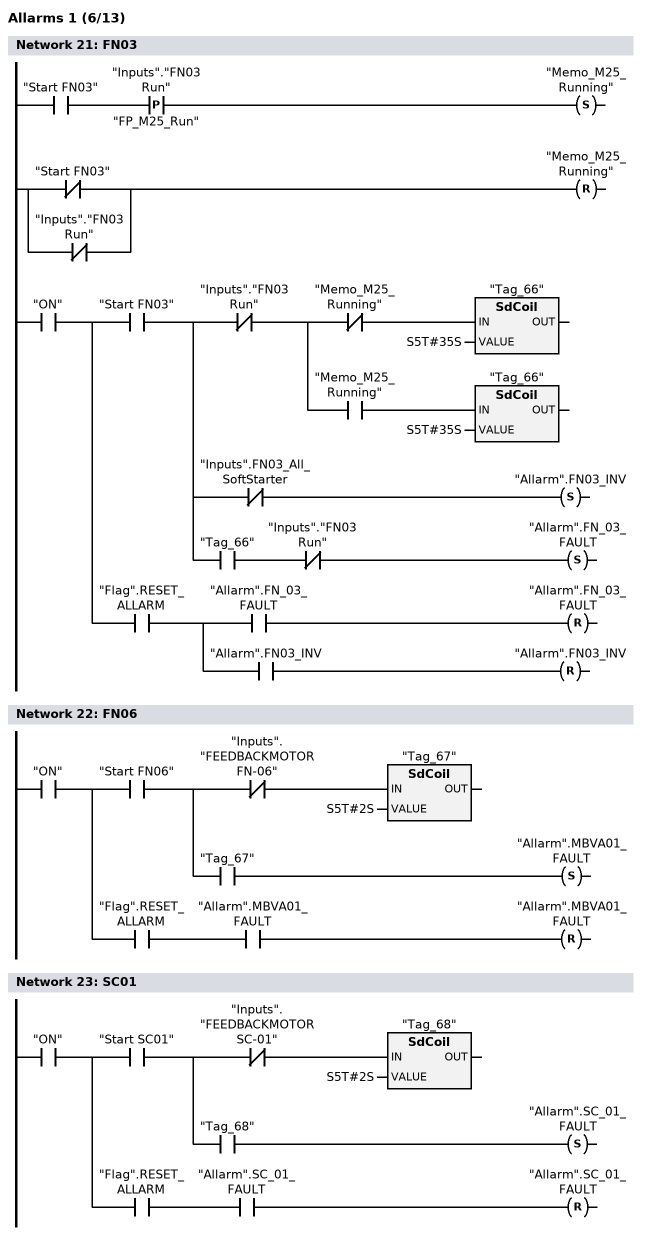
   // no SCL statement known for SdCoil: written as a call
   #_w1 := "Start FN03" AND "Inputs"."FN03 Run" AND NOT "FP_M25_Run";   // rising edge of "Inputs"."FN03 Run"
   "FP_M25_Run" := "Inputs"."FN03 Run";
   IF #_w1 THEN "Memo_M25_Running" := TRUE; END_IF;
   IF NOT "Start FN03" OR NOT "Inputs"."FN03 Run" THEN "Memo_M25_Running" := FALSE; END_IF;
   #_w2 := "ON" AND "Start FN03";
   #_w3 := #_w2 AND NOT "Inputs"."FN03 Run";
   #_w4 := "ON";
   SdCoil(in := #_w3 AND NOT "Memo_M25_Running", value := S5T#35S, operand := "Tag_66");
   SdCoil(in := #_w3 AND "Memo_M25_Running", value := S5T#35S, operand := "Tag_66");
   IF #_w2 AND NOT "Inputs".FN03_All_SoftStarter THEN "Allarm".FN03_INV := TRUE; END_IF;
   IF #_w2 AND "Tag_66" AND NOT "Inputs"."FN03 Run" THEN "Allarm".FN_03_FAULT := TRUE; END_IF;
   #_w5 := #_w4 AND "Flag".RESET_ALLARM;
   IF #_w5 AND "Allarm".FN_03_FAULT THEN "Allarm".FN_03_FAULT := FALSE; END_IF;
   IF #_w5 AND "Allarm".FN03_INV THEN "Allarm".FN03_INV := FALSE; END_IF;
END_REGION

REGION Network 22: FN06
   // no SCL statement known for SdCoil: written as a call
   #_w1 := "ON" AND "Start FN06";
   #_w2 := "ON";
   SdCoil(in := #_w1 AND NOT "Inputs"."FEEDBACKMOTOR FN-06", value := S5T#2S, operand := "Tag_67");
   IF #_w1 AND "Tag_67" THEN "Allarm".MBVA01_FAULT := TRUE; END_IF;
   IF #_w2 AND "Flag".RESET_ALLARM AND "Allarm".MBVA01_FAULT THEN "Allarm".MBVA01_FAULT := FALSE; END_IF;
END_REGION

REGION Network 23: SC01
   // no SCL statement known for SdCoil: written as a call
   #_w1 := "ON" AND "Start SC01";
   #_w2 := "ON";
   SdCoil(in := #_w1 AND NOT "Inputs"."FEEDBACKMOTOR SC-01", value := S5T#2S, operand := "Tag_68");
   IF #_w1 AND "Tag_68" THEN "Allarm".SC_01_FAULT := TRUE; END_IF;
   IF #_w2 AND "Flag".RESET_ALLARM AND "Allarm".SC_01_FAULT THEN "Allarm".SC_01_FAULT := FALSE; END_IF;
END_REGION

REGION Network 24: FN01_FAN DELETED
END_REGION

REGION Network 25: LD01
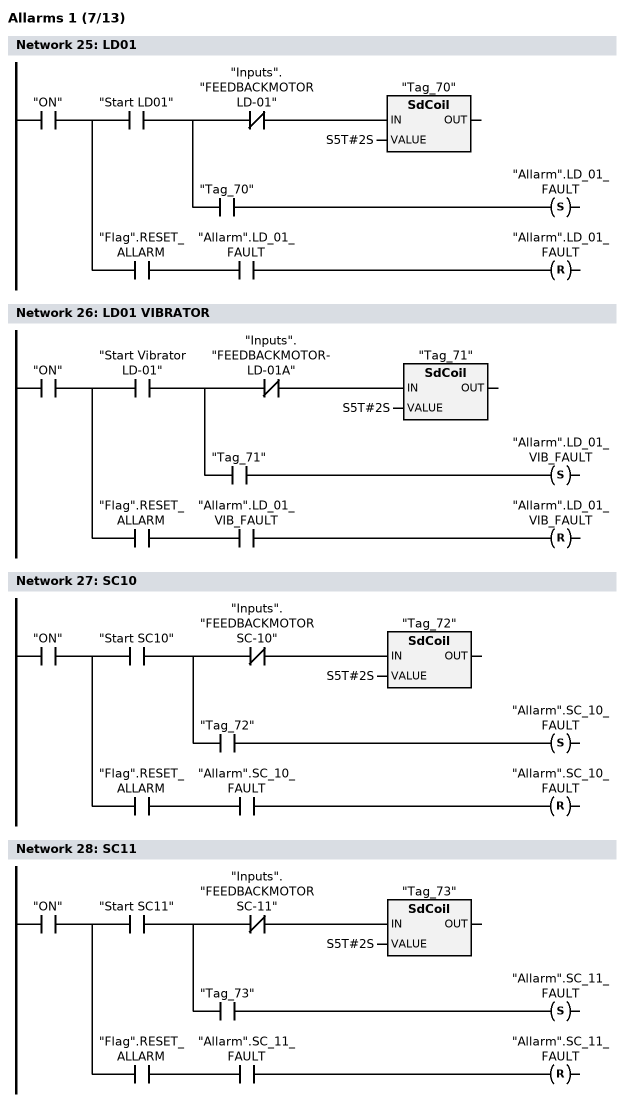
   // no SCL statement known for SdCoil: written as a call
   #_w1 := "ON" AND "Start LD01";
   #_w2 := "ON";
   SdCoil(in := #_w1 AND NOT "Inputs"."FEEDBACKMOTOR LD-01", value := S5T#2S, operand := "Tag_70");
   IF #_w1 AND "Tag_70" THEN "Allarm".LD_01_FAULT := TRUE; END_IF;
   IF #_w2 AND "Flag".RESET_ALLARM AND "Allarm".LD_01_FAULT THEN "Allarm".LD_01_FAULT := FALSE; END_IF;
END_REGION

REGION Network 26: LD01 VIBRATOR
   // no SCL statement known for SdCoil: written as a call
   #_w1 := "ON" AND "Start Vibrator LD-01";
   #_w2 := "ON";
   SdCoil(in := #_w1 AND NOT "Inputs"."FEEDBACKMOTOR-LD-01A", value := S5T#2S, operand := "Tag_71");
   IF #_w1 AND "Tag_71" THEN "Allarm".LD_01_VIB_FAULT := TRUE; END_IF;
   IF #_w2 AND "Flag".RESET_ALLARM AND "Allarm".LD_01_VIB_FAULT THEN
       "Allarm".LD_01_VIB_FAULT := FALSE;
   END_IF;
END_REGION

REGION Network 27: SC10
   // no SCL statement known for SdCoil: written as a call
   #_w1 := "ON" AND "Start SC10";
   #_w2 := "ON";
   SdCoil(in := #_w1 AND NOT "Inputs"."FEEDBACKMOTOR SC-10", value := S5T#2S, operand := "Tag_72");
   IF #_w1 AND "Tag_72" THEN "Allarm".SC_10_FAULT := TRUE; END_IF;
   IF #_w2 AND "Flag".RESET_ALLARM AND "Allarm".SC_10_FAULT THEN "Allarm".SC_10_FAULT := FALSE; END_IF;
END_REGION

REGION Network 28: SC11
   // no SCL statement known for SdCoil: written as a call
   #_w1 := "ON" AND "Start SC11";
   #_w2 := "ON";
   SdCoil(in := #_w1 AND NOT "Inputs"."FEEDBACKMOTOR SC-11", value := S5T#2S, operand := "Tag_73");
   IF #_w1 AND "Tag_73" THEN "Allarm".SC_11_FAULT := TRUE; END_IF;
   IF #_w2 AND "Flag".RESET_ALLARM AND "Allarm".SC_11_FAULT THEN "Allarm".SC_11_FAULT := FALSE; END_IF;
END_REGION

REGION Network 29: FN04
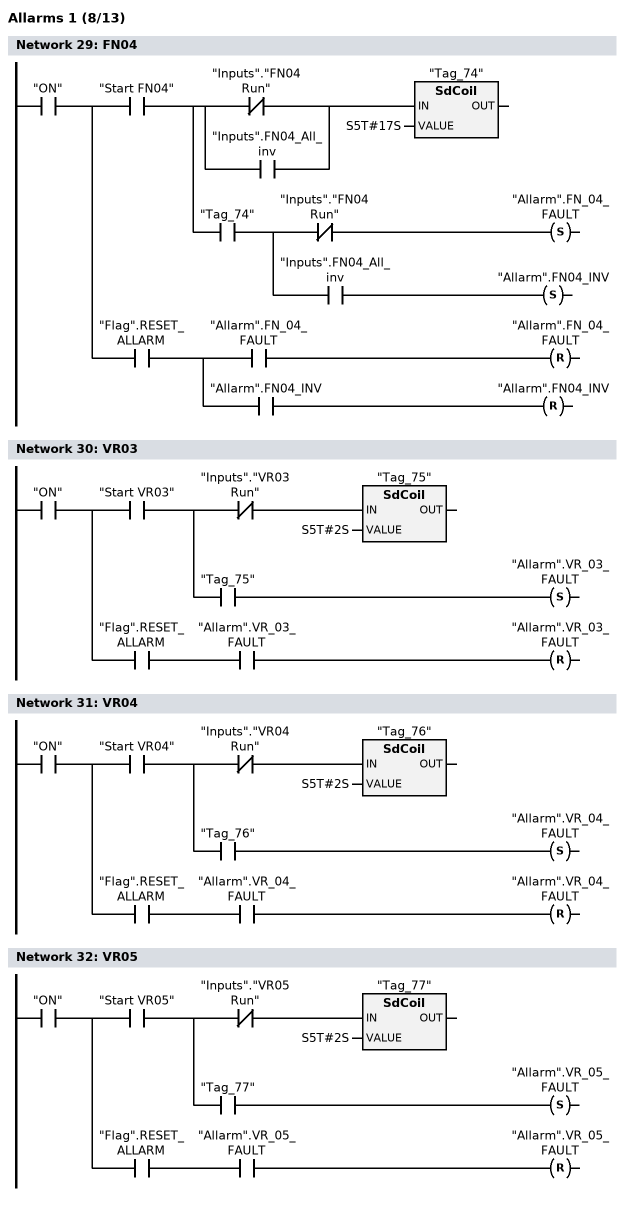
   // no SCL statement known for SdCoil: written as a call
   #_w1 := "ON" AND "Start FN04";
   #_w2 := "ON";
   SdCoil(in := #_w1 AND (NOT "Inputs"."FN04 Run" OR "Inputs".FN04_All_inv),
          value := S5T#17S,
          operand := "Tag_74");
   #_w3 := #_w1 AND "Tag_74";
   IF #_w3 AND NOT "Inputs"."FN04 Run" THEN "Allarm".FN_04_FAULT := TRUE; END_IF;
   IF #_w3 AND "Inputs".FN04_All_inv THEN "Allarm".FN04_INV := TRUE; END_IF;
   #_w4 := #_w2 AND "Flag".RESET_ALLARM;
   IF #_w4 AND "Allarm".FN_04_FAULT THEN "Allarm".FN_04_FAULT := FALSE; END_IF;
   IF #_w4 AND "Allarm".FN04_INV THEN "Allarm".FN04_INV := FALSE; END_IF;
END_REGION

REGION Network 30: VR03
   // no SCL statement known for SdCoil: written as a call
   #_w1 := "ON" AND "Start VR03";
   #_w2 := "ON";
   SdCoil(in := #_w1 AND NOT "Inputs"."VR03 Run", value := S5T#2S, operand := "Tag_75");
   IF #_w1 AND "Tag_75" THEN "Allarm".VR_03_FAULT := TRUE; END_IF;
   IF #_w2 AND "Flag".RESET_ALLARM AND "Allarm".VR_03_FAULT THEN "Allarm".VR_03_FAULT := FALSE; END_IF;
END_REGION

REGION Network 31: VR04
   // no SCL statement known for SdCoil: written as a call
   #_w1 := "ON" AND "Start VR04";
   #_w2 := "ON";
   SdCoil(in := #_w1 AND NOT "Inputs"."VR04 Run", value := S5T#2S, operand := "Tag_76");
   IF #_w1 AND "Tag_76" THEN "Allarm".VR_04_FAULT := TRUE; END_IF;
   IF #_w2 AND "Flag".RESET_ALLARM AND "Allarm".VR_04_FAULT THEN "Allarm".VR_04_FAULT := FALSE; END_IF;
END_REGION

REGION Network 32: VR05
   // no SCL statement known for SdCoil: written as a call
   #_w1 := "ON" AND "Start VR05";
   #_w2 := "ON";
   SdCoil(in := #_w1 AND NOT "Inputs"."VR05 Run", value := S5T#2S, operand := "Tag_77");
   IF #_w1 AND "Tag_77" THEN "Allarm".VR_05_FAULT := TRUE; END_IF;
   IF #_w2 AND "Flag".RESET_ALLARM AND "Allarm".VR_05_FAULT THEN "Allarm".VR_05_FAULT := FALSE; END_IF;
END_REGION

REGION Network 33: VR06
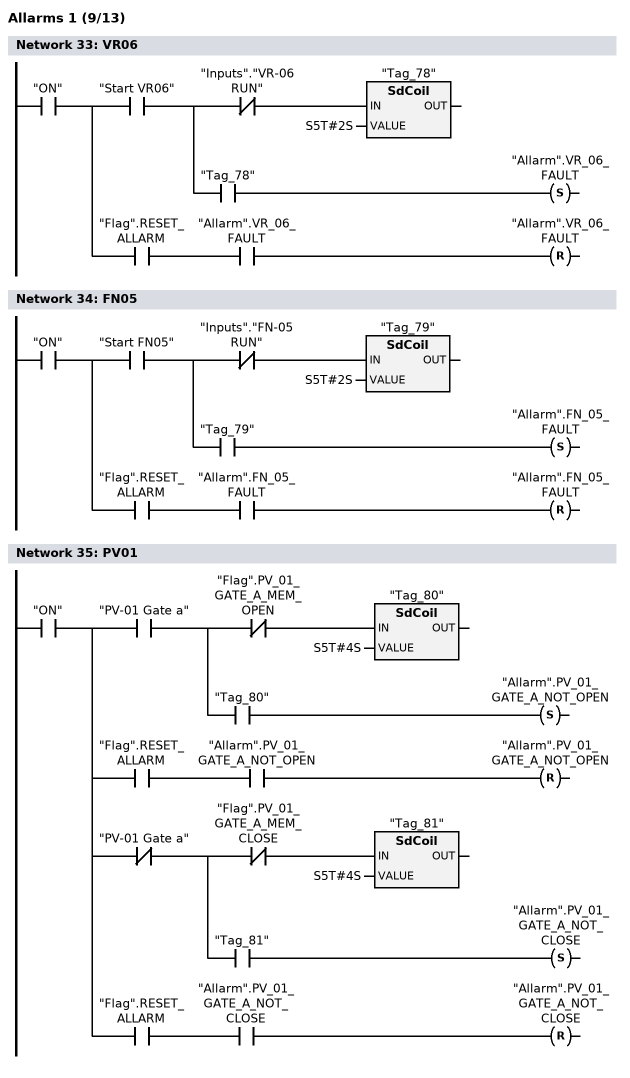
   // no SCL statement known for SdCoil: written as a call
   #_w1 := "ON" AND "Start VR06";
   #_w2 := "ON";
   SdCoil(in := #_w1 AND NOT "Inputs"."VR-06 RUN", value := S5T#2S, operand := "Tag_78");
   IF #_w1 AND "Tag_78" THEN "Allarm".VR_06_FAULT := TRUE; END_IF;
   IF #_w2 AND "Flag".RESET_ALLARM AND "Allarm".VR_06_FAULT THEN "Allarm".VR_06_FAULT := FALSE; END_IF;
END_REGION

REGION Network 34: FN05
   // no SCL statement known for SdCoil: written as a call
   #_w1 := "ON" AND "Start FN05";
   #_w2 := "ON";
   SdCoil(in := #_w1 AND NOT "Inputs"."FN-05 RUN", value := S5T#2S, operand := "Tag_79");
   IF #_w1 AND "Tag_79" THEN "Allarm".FN_05_FAULT := TRUE; END_IF;
   IF #_w2 AND "Flag".RESET_ALLARM AND "Allarm".FN_05_FAULT THEN "Allarm".FN_05_FAULT := FALSE; END_IF;
END_REGION

REGION Network 35: PV01
   // no SCL statement known for SdCoil: written as a call
   #_w1 := "ON" AND "PV-01 Gate a";
   #_w2 := "ON";
   SdCoil(in := #_w1 AND NOT "Flag".PV_01_GATE_A_MEM_OPEN, value := S5T#4S, operand := "Tag_80");
   IF #_w1 AND "Tag_80" THEN "Allarm".PV_01_GATE_A_NOT_OPEN := TRUE; END_IF;
   IF #_w2 AND "Flag".RESET_ALLARM AND "Allarm".PV_01_GATE_A_NOT_OPEN THEN
       "Allarm".PV_01_GATE_A_NOT_OPEN := FALSE;
   END_IF;
   #_w3 := #_w2 AND NOT "PV-01 Gate a";
   SdCoil(in := #_w3 AND NOT "Flag".PV_01_GATE_A_MEM_CLOSE, value := S5T#4S, operand := "Tag_81");
   IF #_w3 AND "Tag_81" THEN "Allarm".PV_01_GATE_A_NOT_CLOSE := TRUE; END_IF;
   IF #_w2 AND "Flag".RESET_ALLARM AND "Allarm".PV_01_GATE_A_NOT_CLOSE THEN
       "Allarm".PV_01_GATE_A_NOT_CLOSE := FALSE;
   END_IF;
END_REGION

REGION Network 36: PV01
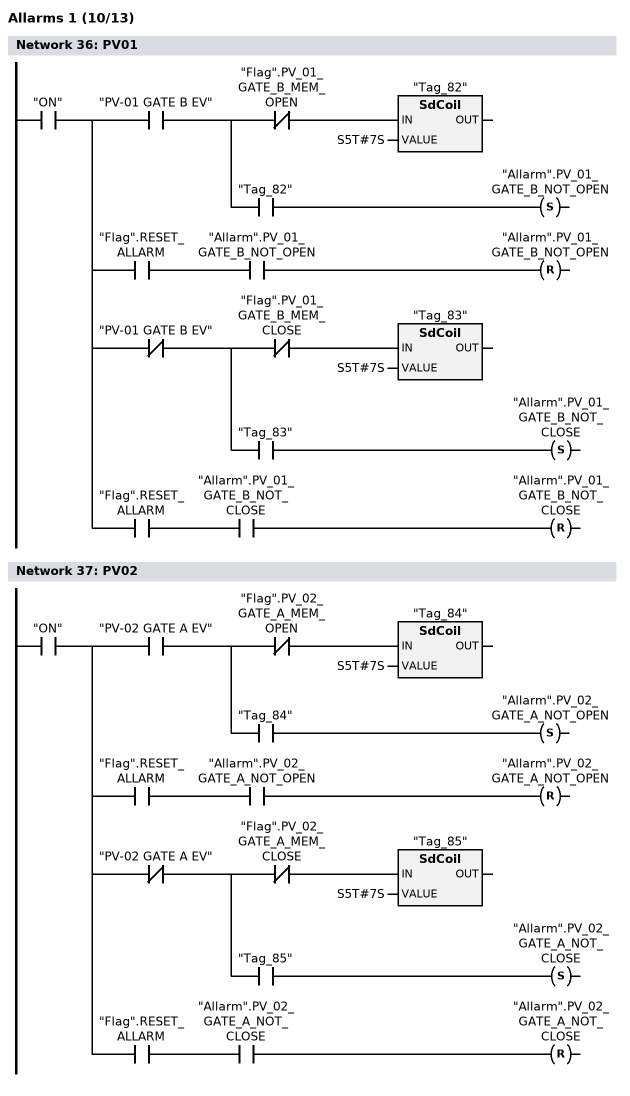
   // no SCL statement known for SdCoil: written as a call
   #_w1 := "ON" AND "PV-01 GATE B EV";
   #_w2 := "ON";
   SdCoil(in := #_w1 AND NOT "Flag".PV_01_GATE_B_MEM_OPEN, value := S5T#7S, operand := "Tag_82");
   IF #_w1 AND "Tag_82" THEN "Allarm".PV_01_GATE_B_NOT_OPEN := TRUE; END_IF;
   IF #_w2 AND "Flag".RESET_ALLARM AND "Allarm".PV_01_GATE_B_NOT_OPEN THEN
       "Allarm".PV_01_GATE_B_NOT_OPEN := FALSE;
   END_IF;
   #_w3 := #_w2 AND NOT "PV-01 GATE B EV";
   SdCoil(in := #_w3 AND NOT "Flag".PV_01_GATE_B_MEM_CLOSE, value := S5T#7S, operand := "Tag_83");
   IF #_w3 AND "Tag_83" THEN "Allarm".PV_01_GATE_B_NOT_CLOSE := TRUE; END_IF;
   IF #_w2 AND "Flag".RESET_ALLARM AND "Allarm".PV_01_GATE_B_NOT_CLOSE THEN
       "Allarm".PV_01_GATE_B_NOT_CLOSE := FALSE;
   END_IF;
END_REGION

REGION Network 37: PV02
   // no SCL statement known for SdCoil: written as a call
   #_w1 := "ON" AND "PV-02 GATE A EV";
   #_w2 := "ON";
   SdCoil(in := #_w1 AND NOT "Flag".PV_02_GATE_A_MEM_OPEN, value := S5T#7S, operand := "Tag_84");
   IF #_w1 AND "Tag_84" THEN "Allarm".PV_02_GATE_A_NOT_OPEN := TRUE; END_IF;
   IF #_w2 AND "Flag".RESET_ALLARM AND "Allarm".PV_02_GATE_A_NOT_OPEN THEN
       "Allarm".PV_02_GATE_A_NOT_OPEN := FALSE;
   END_IF;
   #_w3 := #_w2 AND NOT "PV-02 GATE A EV";
   SdCoil(in := #_w3 AND NOT "Flag".PV_02_GATE_A_MEM_CLOSE, value := S5T#7S, operand := "Tag_85");
   IF #_w3 AND "Tag_85" THEN "Allarm".PV_02_GATE_A_NOT_CLOSE := TRUE; END_IF;
   IF #_w2 AND "Flag".RESET_ALLARM AND "Allarm".PV_02_GATE_A_NOT_CLOSE THEN
       "Allarm".PV_02_GATE_A_NOT_CLOSE := FALSE;
   END_IF;
END_REGION

REGION Network 38: PV02
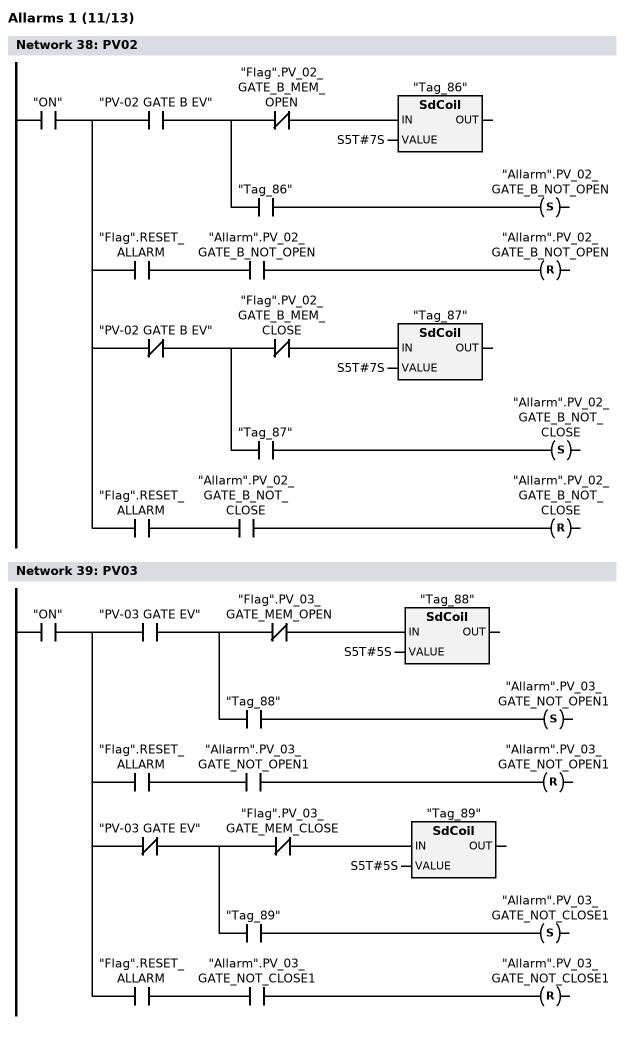
   // no SCL statement known for SdCoil: written as a call
   #_w1 := "ON" AND "PV-02 GATE B EV";
   #_w2 := "ON";
   SdCoil(in := #_w1 AND NOT "Flag".PV_02_GATE_B_MEM_OPEN, value := S5T#7S, operand := "Tag_86");
   IF #_w1 AND "Tag_86" THEN "Allarm".PV_02_GATE_B_NOT_OPEN := TRUE; END_IF;
   IF #_w2 AND "Flag".RESET_ALLARM AND "Allarm".PV_02_GATE_B_NOT_OPEN THEN
       "Allarm".PV_02_GATE_B_NOT_OPEN := FALSE;
   END_IF;
   #_w3 := #_w2 AND NOT "PV-02 GATE B EV";
   SdCoil(in := #_w3 AND NOT "Flag".PV_02_GATE_B_MEM_CLOSE, value := S5T#7S, operand := "Tag_87");
   IF #_w3 AND "Tag_87" THEN "Allarm".PV_02_GATE_B_NOT_CLOSE := TRUE; END_IF;
   IF #_w2 AND "Flag".RESET_ALLARM AND "Allarm".PV_02_GATE_B_NOT_CLOSE THEN
       "Allarm".PV_02_GATE_B_NOT_CLOSE := FALSE;
   END_IF;
END_REGION

REGION Network 39: PV03
   // no SCL statement known for SdCoil: written as a call
   #_w1 := "ON" AND "PV-03 GATE EV";
   #_w2 := "ON";
   SdCoil(in := #_w1 AND NOT "Flag".PV_03_GATE_MEM_OPEN, value := S5T#5S, operand := "Tag_88");
   IF #_w1 AND "Tag_88" THEN "Allarm".PV_03_GATE_NOT_OPEN1 := TRUE; END_IF;
   IF #_w2 AND "Flag".RESET_ALLARM AND "Allarm".PV_03_GATE_NOT_OPEN1 THEN
       "Allarm".PV_03_GATE_NOT_OPEN1 := FALSE;
   END_IF;
   #_w3 := #_w2 AND NOT "PV-03 GATE EV";
   SdCoil(in := #_w3 AND NOT "Flag".PV_03_GATE_MEM_CLOSE, value := S5T#5S, operand := "Tag_89");
   IF #_w3 AND "Tag_89" THEN "Allarm".PV_03_GATE_NOT_CLOSE1 := TRUE; END_IF;
   IF #_w2 AND "Flag".RESET_ALLARM AND "Allarm".PV_03_GATE_NOT_CLOSE1 THEN
       "Allarm".PV_03_GATE_NOT_CLOSE1 := FALSE;
   END_IF;
END_REGION

REGION Network 40: BWF01/BWF02
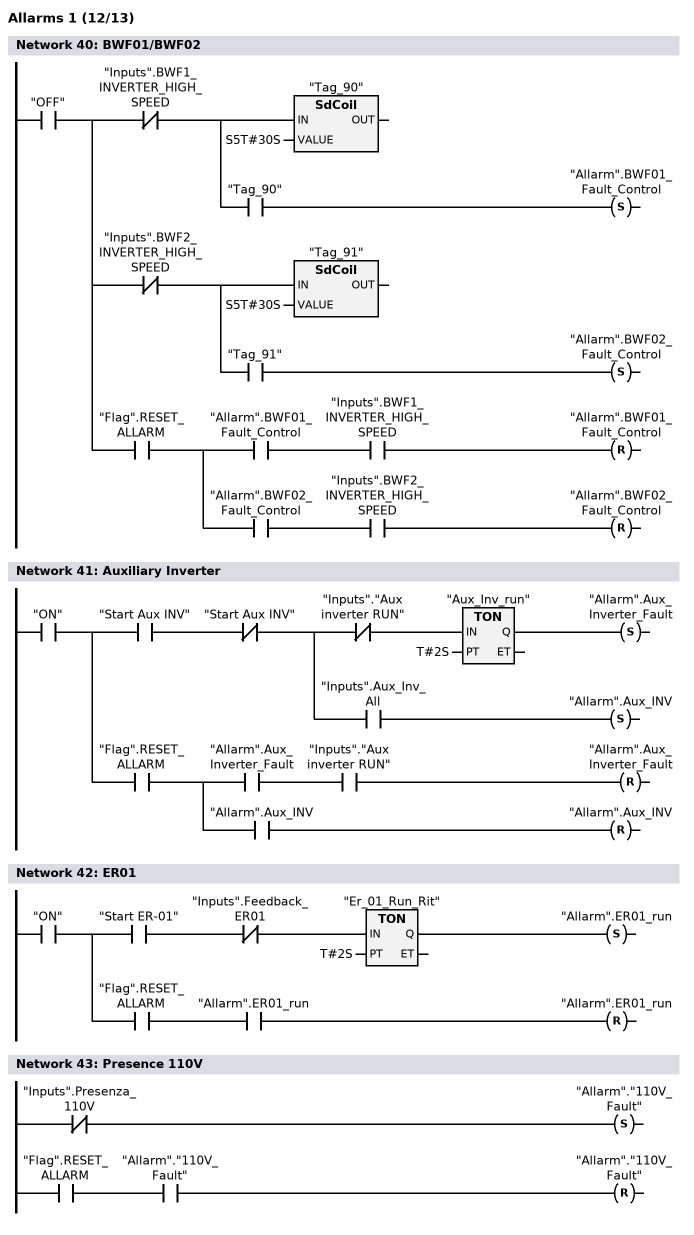
   // no SCL statement known for SdCoil: written as a call
   #_w1 := "OFF" AND NOT "Inputs".BWF1_INVERTER_HIGH_SPEED;
   #_w2 := "OFF";
   SdCoil(in := #_w1, value := S5T#30S, operand := "Tag_90");
   IF #_w1 AND "Tag_90" THEN "Allarm".BWF01_Fault_Control := TRUE; END_IF;
   #_w3 := #_w2 AND NOT "Inputs".BWF2_INVERTER_HIGH_SPEED;
   SdCoil(in := #_w3, value := S5T#30S, operand := "Tag_91");
   IF #_w3 AND "Tag_91" THEN "Allarm".BWF02_Fault_Control := TRUE; END_IF;
   #_w4 := #_w2 AND "Flag".RESET_ALLARM;
   IF #_w4 AND "Allarm".BWF01_Fault_Control AND "Inputs".BWF1_INVERTER_HIGH_SPEED THEN
       "Allarm".BWF01_Fault_Control := FALSE;
   END_IF;
   IF #_w4 AND "Allarm".BWF02_Fault_Control AND "Inputs".BWF2_INVERTER_HIGH_SPEED THEN
       "Allarm".BWF02_Fault_Control := FALSE;
   END_IF;
END_REGION

REGION Network 41: Auxiliary Inverter
   #_w1 := "ON" AND "Start Aux INV" AND NOT "Start Aux INV";
   "Aux_Inv_run".TON(IN := #_w1 AND NOT "Inputs"."Aux inverter RUN", PT := T#2S);
   IF "Aux_Inv_run".Q THEN "Allarm".Aux_Inverter_Fault := TRUE; END_IF;
   IF #_w1 AND "Inputs".Aux_Inv_All THEN "Allarm".Aux_INV := TRUE; END_IF;
   #_w2 := "ON" AND "Flag".RESET_ALLARM;
   IF #_w2 AND "Allarm".Aux_Inverter_Fault AND "Inputs"."Aux inverter RUN" THEN
       "Allarm".Aux_Inverter_Fault := FALSE;
   END_IF;
   IF #_w2 AND "Allarm".Aux_INV THEN "Allarm".Aux_INV := FALSE; END_IF;
END_REGION

REGION Network 42: ER01
   "Er_01_Run_Rit".TON(IN := "ON" AND "Start ER-01" AND NOT "Inputs".Feedback_ER01, PT := T#2S);
   IF "Er_01_Run_Rit".Q THEN "Allarm".ER01_run := TRUE; END_IF;
   IF "ON" AND "Flag".RESET_ALLARM AND "Allarm".ER01_run THEN "Allarm".ER01_run := FALSE; END_IF;
END_REGION

REGION Network 43: Presence 110V
   RUNG wire#powerrail
      I_Contact( "Inputs".Presenza_110V )
      S_Coil( "Allarm"."110V_Fault" )
   END_RUNG
   RUNG wire#powerrail
      Contact( "Flag".RESET_ALLARM )
      Contact( "Allarm"."110V_Fault" )
      R_Coil( "Allarm"."110V_Fault" )
   END_RUNG
   // the same network as SCL:
   IF NOT "Inputs".Presenza_110V THEN "Allarm"."110V_Fault" := TRUE; END_IF;
   IF "Flag".RESET_ALLARM AND "Allarm"."110V_Fault" THEN "Allarm"."110V_Fault" := FALSE; END_IF;
END_REGION

REGION Network 44: Module emergenzy OK
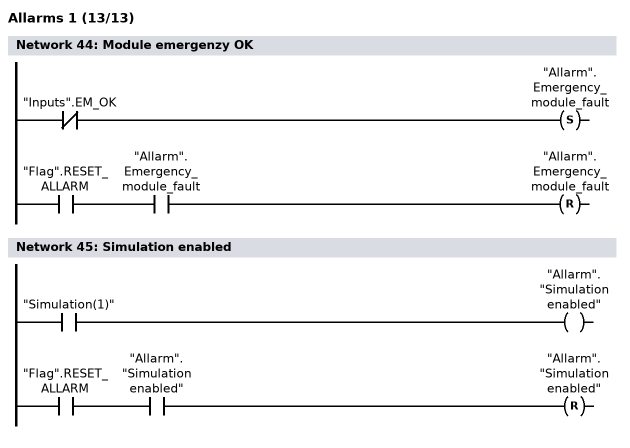
   RUNG wire#powerrail
      I_Contact( "Inputs".EM_OK )
      S_Coil( "Allarm".Emergency_module_fault )
   END_RUNG
   RUNG wire#powerrail
      Contact( "Flag".RESET_ALLARM )
      Contact( "Allarm".Emergency_module_fault )
      R_Coil( "Allarm".Emergency_module_fault )
   END_RUNG
   // the same network as SCL:
   IF NOT "Inputs".EM_OK THEN "Allarm".Emergency_module_fault := TRUE; END_IF;
   IF "Flag".RESET_ALLARM AND "Allarm".Emergency_module_fault THEN
       "Allarm".Emergency_module_fault := FALSE;
   END_IF;
END_REGION

REGION Network 45: Simulation enabled
   RUNG wire#powerrail
      Contact( "Simulation(1)" )
      Coil( "Allarm"."Simulation enabled" )
   END_RUNG
   RUNG wire#powerrail
      Contact( "Flag".RESET_ALLARM )
      Contact( "Allarm"."Simulation enabled" )
      R_Coil( "Allarm"."Simulation enabled" )
   END_RUNG
   // the same network as SCL:
   "Allarm"."Simulation enabled" := "Simulation(1)";
   IF "Flag".RESET_ALLARM AND "Allarm"."Simulation enabled" THEN
       "Allarm"."Simulation enabled" := FALSE;
   END_IF;
END_REGION
END_FUNCTION

FUNCTION "Allarms 2" : Void   // FC5, LAD
{ S7_Optimized_Access := 'FALSE' }
VERSION : 0.1
   VAR_TEMP
      APP : Int;
   END_VAR
   VAR_TEMP   // added for the SCL form of the ladder/FBD networks
      _w1 : Bool;
      _w2 : Bool;
      _w3 : Bool;
      _w4 : Bool;
      _w5 : Bool;
      _w6 : Bool;
      _w7 : Bool;
   END_VAR
BEGIN

REGION Network 1: Motorized butterfly valves / MV-01 Motorized valve fault
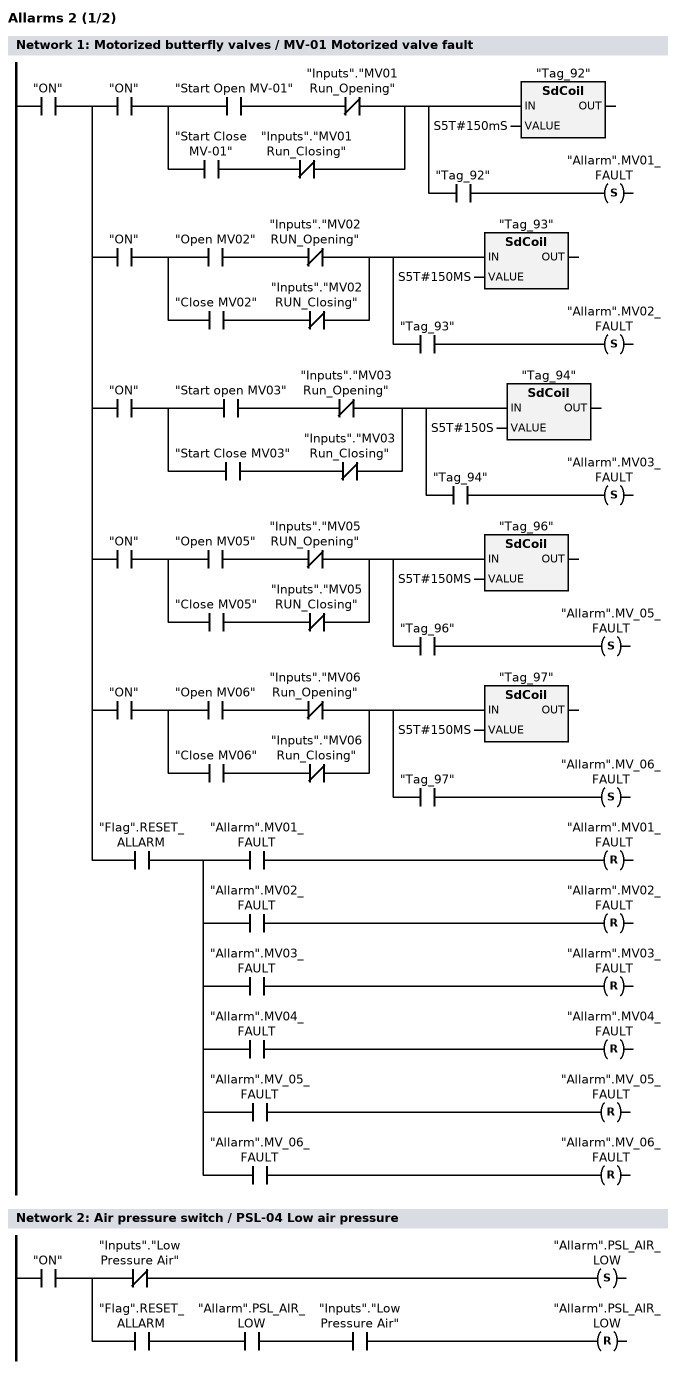
   // no SCL statement known for SdCoil: written as a call
   #_w1 := "ON" AND "ON" AND (("Start Open MV-01" AND NOT "Inputs"."MV01 Run_Opening") OR ("Start Close MV-01" AND NOT "Inputs"."MV01 Run_Closing"));
   #_w2 := "ON";
   SdCoil(in := #_w1, value := S5T#150mS, operand := "Tag_92");
   IF #_w1 AND "Tag_92" THEN "Allarm".MV01_FAULT := TRUE; END_IF;
   #_w3 := #_w2 AND "ON" AND (("Open MV02" AND NOT "Inputs"."MV02 RUN_Opening") OR ("Close MV02" AND NOT "Inputs"."MV02 RUN_Closing"));
   SdCoil(in := #_w3, value := S5T#150MS, operand := "Tag_93");
   IF #_w3 AND "Tag_93" THEN "Allarm".MV02_FAULT := TRUE; END_IF;
   #_w4 := #_w2 AND "ON" AND (("Start open MV03" AND NOT "Inputs"."MV03 Run_Opening") OR ("Start Close MV03" AND NOT "Inputs"."MV03 Run_Closing"));
   SdCoil(in := #_w4, value := S5T#150S, operand := "Tag_94");
   IF #_w4 AND "Tag_94" THEN "Allarm".MV03_FAULT := TRUE; END_IF;
   #_w5 := #_w2 AND "ON" AND (("Open MV05" AND NOT "Inputs"."MV05 RUN_Opening") OR ("Close MV05" AND NOT "Inputs"."MV05 RUN_Closing"));
   SdCoil(in := #_w5, value := S5T#150MS, operand := "Tag_96");
   IF #_w5 AND "Tag_96" THEN "Allarm".MV_05_FAULT := TRUE; END_IF;
   #_w6 := #_w2 AND "ON" AND (("Open MV06" AND NOT "Inputs"."MV06 Run_Opening") OR ("Close MV06" AND NOT "Inputs"."MV06 Run_Closing"));
   SdCoil(in := #_w6, value := S5T#150MS, operand := "Tag_97");
   IF #_w6 AND "Tag_97" THEN "Allarm".MV_06_FAULT := TRUE; END_IF;
   #_w7 := #_w2 AND "Flag".RESET_ALLARM;
   IF #_w7 AND "Allarm".MV01_FAULT THEN "Allarm".MV01_FAULT := FALSE; END_IF;
   IF #_w7 AND "Allarm".MV02_FAULT THEN "Allarm".MV02_FAULT := FALSE; END_IF;
   IF #_w7 AND "Allarm".MV03_FAULT THEN "Allarm".MV03_FAULT := FALSE; END_IF;
   IF #_w7 AND "Allarm".MV04_FAULT THEN "Allarm".MV04_FAULT := FALSE; END_IF;
   IF #_w7 AND "Allarm".MV_05_FAULT THEN "Allarm".MV_05_FAULT := FALSE; END_IF;
   IF #_w7 AND "Allarm".MV_06_FAULT THEN "Allarm".MV_06_FAULT := FALSE; END_IF;
END_REGION

REGION Network 2: Air pressure switch / PSL-04 Low air pressure
   RUNG wire#powerrail
      Contact( "ON" )
      wire#w1
      I_Contact( "Inputs"."Low Pressure Air" )
      S_Coil( "Allarm".PSL_AIR_LOW )
   END_RUNG
   RUNG wire#w1
      Contact( "Flag".RESET_ALLARM )
      Contact( "Allarm".PSL_AIR_LOW )
      Contact( "Inputs"."Low Pressure Air" )
      R_Coil( "Allarm".PSL_AIR_LOW )
   END_RUNG
   // the same network as SCL:
   IF "ON" AND NOT "Inputs"."Low Pressure Air" THEN "Allarm".PSL_AIR_LOW := TRUE; END_IF;
   IF "ON" AND "Flag".RESET_ALLARM AND "Allarm".PSL_AIR_LOW AND "Inputs"."Low Pressure Air" THEN
       "Allarm".PSL_AIR_LOW := FALSE;
   END_IF;
END_REGION

REGION Network 3: Lime level indicator / LD-01 Low lime level
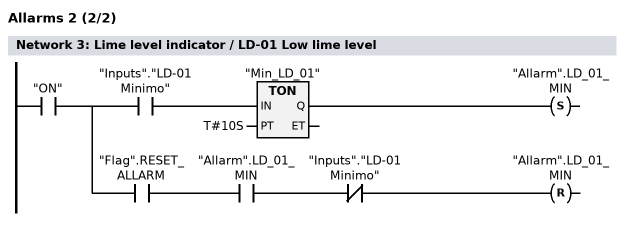
   "Min_LD_01".TON(IN := "ON" AND "Inputs"."LD-01 Minimo", PT := T#10S);
   IF "Min_LD_01".Q THEN "Allarm".LD_01_MIN := TRUE; END_IF;
   IF "ON" AND "Flag".RESET_ALLARM AND "Allarm".LD_01_MIN AND NOT "Inputs"."LD-01 Minimo" THEN
       "Allarm".LD_01_MIN := FALSE;
   END_IF;
END_REGION

REGION Network 4: PV-04 limit SWITCH / PV-04 limit SWITCH DELETED
END_REGION

REGION Network 5: Allarme Valvola PV-04 / Allarm valve PV-04 DELETED
END_REGION
END_FUNCTION

FUNCTION "Allarms 3" : Void   // FC6, LAD
{ S7_Optimized_Access := 'FALSE' }
VERSION : 0.1
   VAR_TEMP
      app00 : Int;
      app01 : Int;
      app02 : Int;
      max_max_tc1 : Int;
      max_max_tc3 : Int;
      max_max_tc6 : Int;
      app03 : Int;
      app04 : Int;
      app05 : Int;
      app06 : Int;
      app07 : Int;
      Somma_Perc_alim : Int;
   END_VAR
   VAR_TEMP   // added for the SCL form of the ladder/FBD networks
      _w1 : Bool;
      _w2 : Bool;
      _w3 : Bool;
      _w4 : Bool;
      _w5 : Bool;
      _w6 : Bool;
   END_VAR
BEGIN

REGION Network 1: MAX TC01 temperature
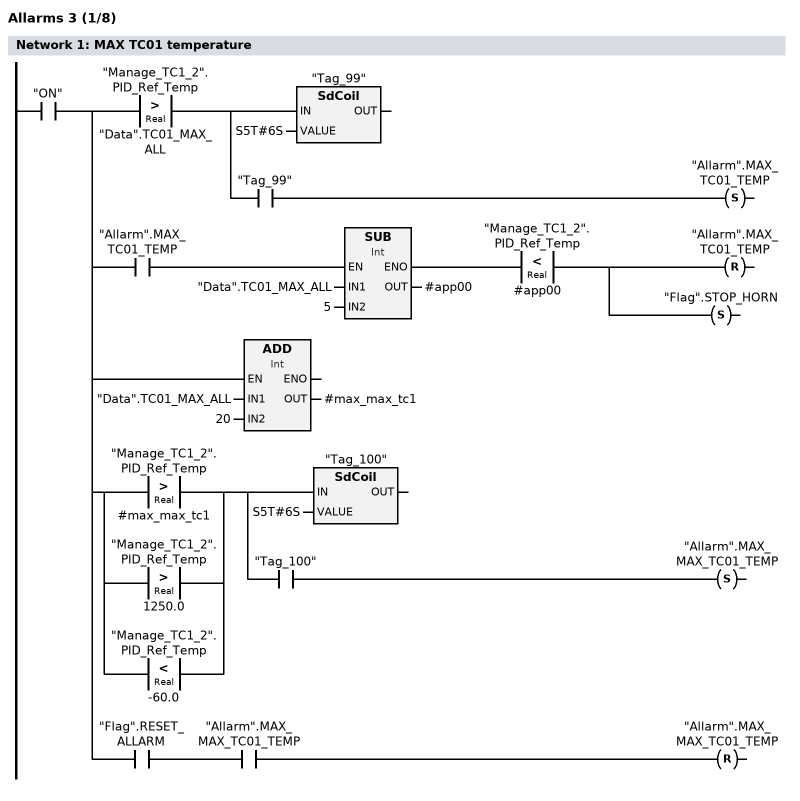
   // no SCL statement known for SdCoil: written as a call
   // ENO of a box is taken as its EN; it also drops when the box reports an error
   #_w1 := "ON" AND ("Manage_TC1_2".PID_Ref_Temp > "Data".TC01_MAX_ALL);
   #_w2 := "ON";
   SdCoil(in := #_w1, value := S5T#6S, operand := "Tag_99");
   IF #_w1 AND "Tag_99" THEN "Allarm".MAX_TC01_TEMP := TRUE; END_IF;
   #_w3 := #_w2 AND "Allarm".MAX_TC01_TEMP;
   IF #_w3 THEN #app00 := "Data".TC01_MAX_ALL - 5; END_IF;
   IF #_w3 AND ("Manage_TC1_2".PID_Ref_Temp < #app00) THEN
       "Allarm".MAX_TC01_TEMP := FALSE;
       "Flag".STOP_HORN := TRUE;
   END_IF;
   IF #_w2 THEN #max_max_tc1 := "Data".TC01_MAX_ALL + 20; END_IF;
   #_w4 := #_w2 AND (("Manage_TC1_2".PID_Ref_Temp > #max_max_tc1) OR ("Manage_TC1_2".PID_Ref_Temp > 1250.0) OR ("Manage_TC1_2".PID_Ref_Temp < (-60.0)));
   SdCoil(in := #_w4, value := S5T#6S, operand := "Tag_100");
   IF #_w4 AND "Tag_100" THEN "Allarm".MAX_MAX_TC01_TEMP := TRUE; END_IF;
   IF #_w2 AND "Flag".RESET_ALLARM AND "Allarm".MAX_MAX_TC01_TEMP THEN
       "Allarm".MAX_MAX_TC01_TEMP := FALSE;
   END_IF;
END_REGION

REGION Network 2: Low TC03 temperature
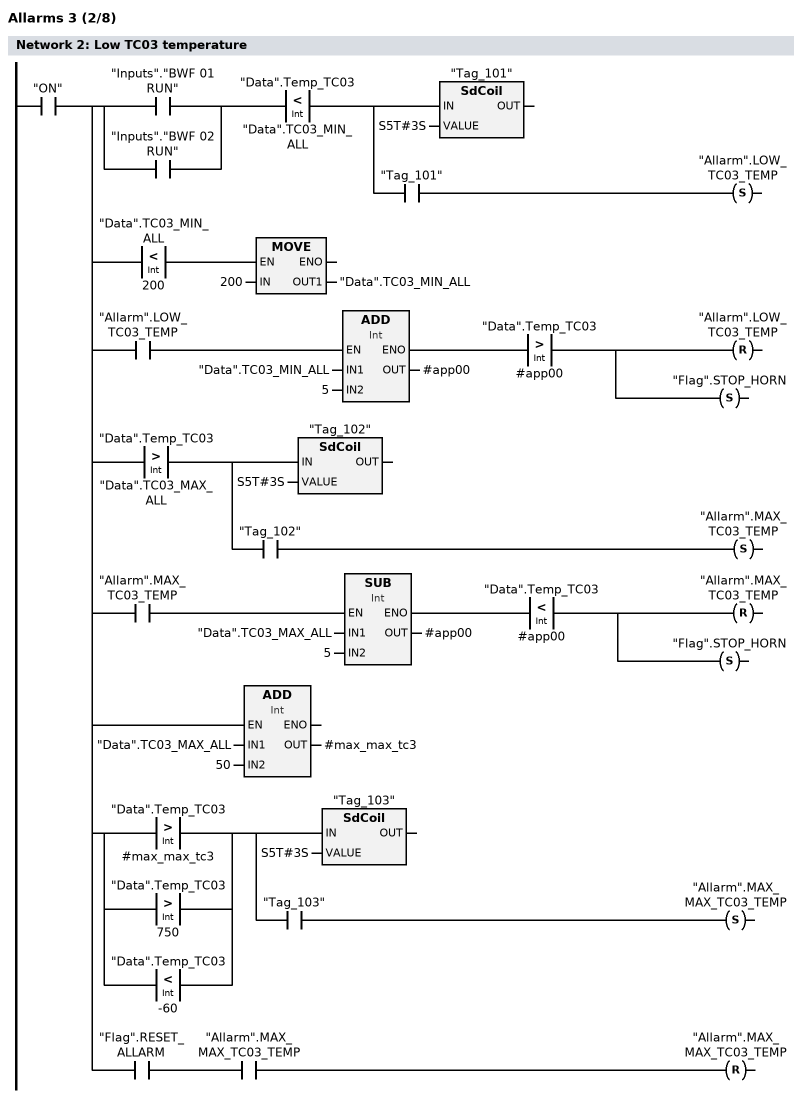
   // no SCL statement known for SdCoil: written as a call
   // ENO of a box is taken as its EN; it also drops when the box reports an error
   #_w1 := "ON" AND ("Inputs"."BWF 01 RUN" OR "Inputs"."BWF 02 RUN") AND ("Data".Temp_TC03 < "Data".TC03_MIN_ALL);
   #_w2 := "ON";
   SdCoil(in := #_w1, value := S5T#3S, operand := "Tag_101");
   IF #_w1 AND "Tag_101" THEN "Allarm".LOW_TC03_TEMP := TRUE; END_IF;
   IF #_w2 AND ("Data".TC03_MIN_ALL < 200) THEN "Data".TC03_MIN_ALL := 200; END_IF;
   #_w3 := #_w2 AND "Allarm".LOW_TC03_TEMP;
   IF #_w3 THEN #app00 := "Data".TC03_MIN_ALL + 5; END_IF;
   IF #_w3 AND ("Data".Temp_TC03 > #app00) THEN
       "Allarm".LOW_TC03_TEMP := FALSE;
       "Flag".STOP_HORN := TRUE;
   END_IF;
   #_w4 := #_w2 AND ("Data".Temp_TC03 > "Data".TC03_MAX_ALL);
   SdCoil(in := #_w4, value := S5T#3S, operand := "Tag_102");
   IF #_w4 AND "Tag_102" THEN "Allarm".MAX_TC03_TEMP := TRUE; END_IF;
   #_w5 := #_w2 AND "Allarm".MAX_TC03_TEMP;
   IF #_w5 THEN #app00 := "Data".TC03_MAX_ALL - 5; END_IF;
   IF #_w5 AND ("Data".Temp_TC03 < #app00) THEN
       "Allarm".MAX_TC03_TEMP := FALSE;
       "Flag".STOP_HORN := TRUE;
   END_IF;
   IF #_w2 THEN #max_max_tc3 := "Data".TC03_MAX_ALL + 50; END_IF;
   #_w6 := #_w2 AND (("Data".Temp_TC03 > #max_max_tc3) OR ("Data".Temp_TC03 > 750) OR ("Data".Temp_TC03 < (-60)));
   SdCoil(in := #_w6, value := S5T#3S, operand := "Tag_103");
   IF #_w6 AND "Tag_103" THEN "Allarm".MAX_MAX_TC03_TEMP := TRUE; END_IF;
   IF #_w2 AND "Flag".RESET_ALLARM AND "Allarm".MAX_MAX_TC03_TEMP THEN
       "Allarm".MAX_MAX_TC03_TEMP := FALSE;
   END_IF;
END_REGION

REGION Network 3: MAX TC04 temperature
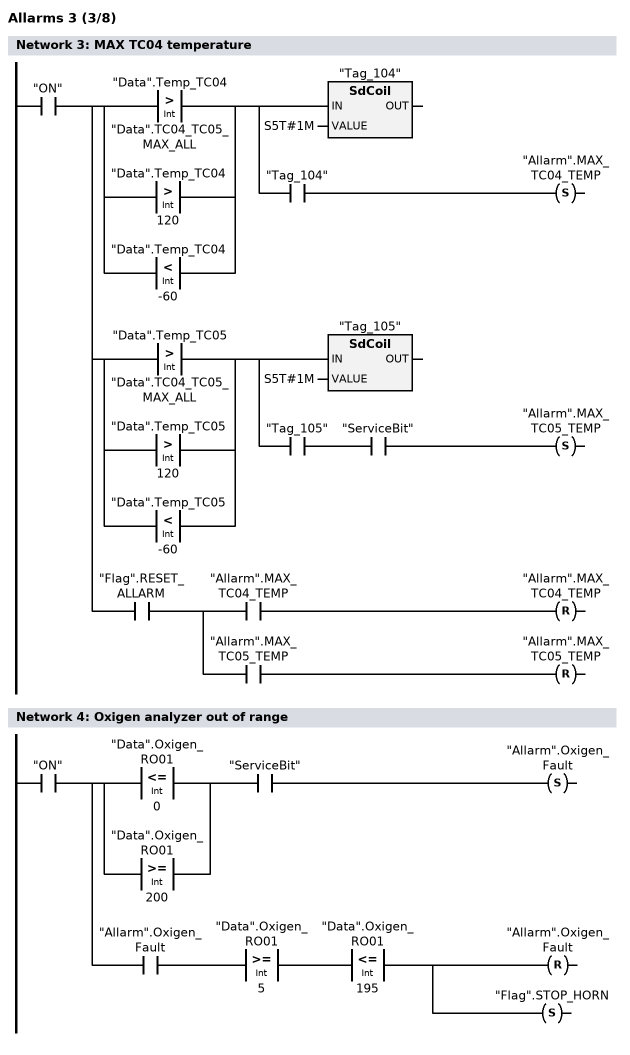
   // no SCL statement known for SdCoil: written as a call
   #_w1 := "ON" AND (("Data".Temp_TC04 > "Data".TC04_TC05_MAX_ALL) OR ("Data".Temp_TC04 > 120) OR ("Data".Temp_TC04 < (-60)));
   #_w2 := "ON";
   SdCoil(in := #_w1, value := S5T#1M, operand := "Tag_104");
   IF #_w1 AND "Tag_104" THEN "Allarm".MAX_TC04_TEMP := TRUE; END_IF;
   #_w3 := #_w2 AND (("Data".Temp_TC05 > "Data".TC04_TC05_MAX_ALL) OR ("Data".Temp_TC05 > 120) OR ("Data".Temp_TC05 < (-60)));
   SdCoil(in := #_w3, value := S5T#1M, operand := "Tag_105");
   IF #_w3 AND "Tag_105" AND "ServiceBit" THEN "Allarm".MAX_TC05_TEMP := TRUE; END_IF;
   #_w4 := #_w2 AND "Flag".RESET_ALLARM;
   IF #_w4 AND "Allarm".MAX_TC04_TEMP THEN "Allarm".MAX_TC04_TEMP := FALSE; END_IF;
   IF #_w4 AND "Allarm".MAX_TC05_TEMP THEN "Allarm".MAX_TC05_TEMP := FALSE; END_IF;
END_REGION

REGION Network 4: Oxigen analyzer out of range
   RUNG wire#powerrail
      Contact( "ON" )
      wire#w1
      { S7_Templates := "SrcType := Int" } LE_Contact(in1 := "Data".Oxigen_RO01, in2 := 0)
      wire#w2
      Contact( "ServiceBit" )
      S_Coil( "Allarm".Oxigen_Fault )
   END_RUNG
   RUNG wire#w1
      { S7_Templates := "SrcType := Int" } GE_Contact(in1 := "Data".Oxigen_RO01, in2 := 200)
   END_RUNG wire#w2
   RUNG wire#w1
      Contact( "Allarm".Oxigen_Fault )
      { S7_Templates := "SrcType := Int" } GE_Contact(in1 := "Data".Oxigen_RO01, in2 := 5)
      { S7_Templates := "SrcType := Int" } LE_Contact(in1 := "Data".Oxigen_RO01, in2 := 195)
      wire#w3
      R_Coil( "Allarm".Oxigen_Fault )
   END_RUNG
   RUNG wire#w3
      S_Coil( "Flag".STOP_HORN )
   END_RUNG
   // the same network as SCL:
   IF "ON" AND (("Data".Oxigen_RO01 <= 0) OR ("Data".Oxigen_RO01 >= 200)) AND "ServiceBit" THEN
       "Allarm".Oxigen_Fault := TRUE;
   END_IF;
   #_w1 := "ON" AND "Allarm".Oxigen_Fault AND ("Data".Oxigen_RO01 >= 5) AND ("Data".Oxigen_RO01 <= 195);
   IF #_w1 THEN
       "Allarm".Oxigen_Fault := FALSE;
       "Flag".STOP_HORN := TRUE;
   END_IF;
END_REGION

REGION Network 5: Oxigen too high
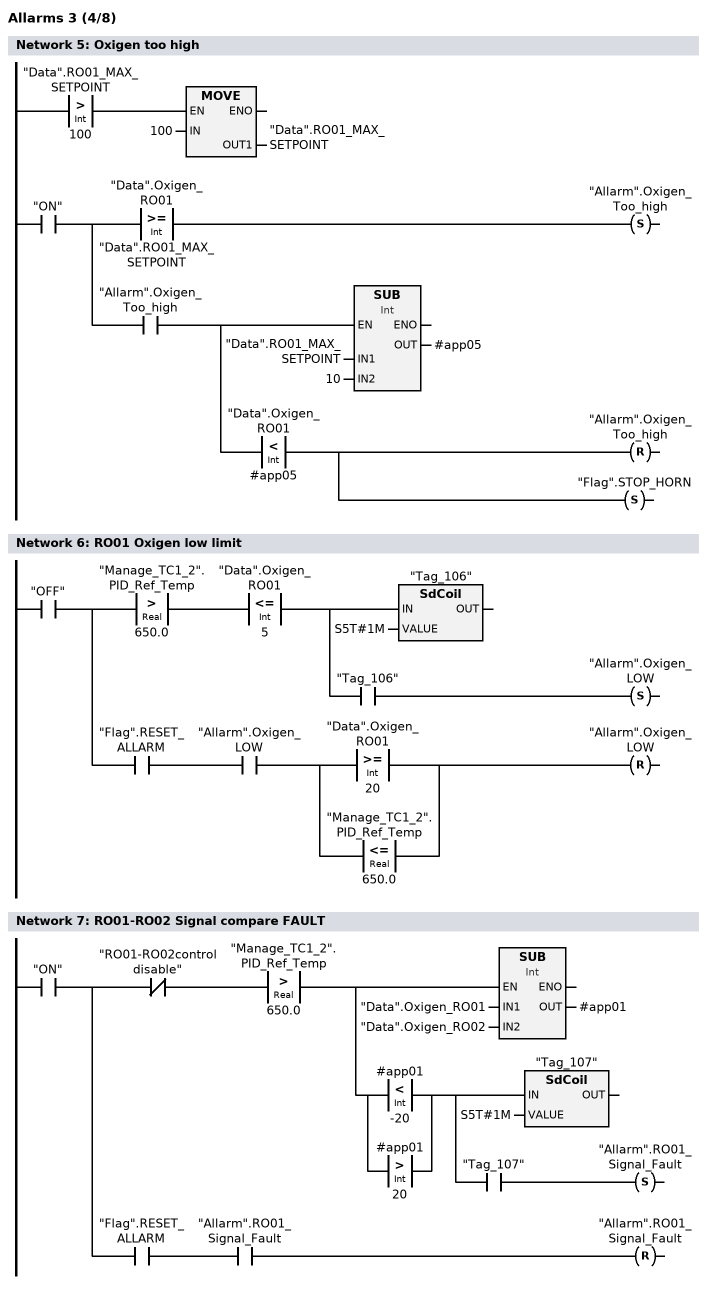
   RUNG wire#powerrail
      { S7_Templates := "SrcType := Int" } GT_Contact(in1 := "Data".RO01_MAX_SETPOINT, in2 := 100)
      Move(in := 100, out1 => "Data".RO01_MAX_SETPOINT)
   END_RUNG
   RUNG wire#powerrail
      Contact( "ON" )
      wire#w1
      { S7_Templates := "SrcType := Int" } GE_Contact(in1 := "Data".Oxigen_RO01, in2 := "Data".RO01_MAX_SETPOINT)
      S_Coil( "Allarm".Oxigen_Too_high )
   END_RUNG
   RUNG wire#w1
      Contact( "Allarm".Oxigen_Too_high )
      wire#w2
      { S7_Templates := "SrcType := Int"; S7_GenerateENO := "TRUE" } Sub(in1 := "Data".RO01_MAX_SETPOINT, in2 := 10, out => #app05)
   END_RUNG
   RUNG wire#w2
      { S7_Templates := "SrcType := Int" } LT_Contact(in1 := "Data".Oxigen_RO01, in2 := #app05)
      wire#w3
      R_Coil( "Allarm".Oxigen_Too_high )
   END_RUNG
   RUNG wire#w3
      S_Coil( "Flag".STOP_HORN )
   END_RUNG
   // the same network as SCL:
   IF "Data".RO01_MAX_SETPOINT > 100 THEN "Data".RO01_MAX_SETPOINT := 100; END_IF;
   IF "ON" AND ("Data".Oxigen_RO01 >= "Data".RO01_MAX_SETPOINT) THEN
       "Allarm".Oxigen_Too_high := TRUE;
   END_IF;
   #_w1 := "ON" AND "Allarm".Oxigen_Too_high;
   IF #_w1 THEN #app05 := "Data".RO01_MAX_SETPOINT - 10; END_IF;
   IF #_w1 AND ("Data".Oxigen_RO01 < #app05) THEN
       "Allarm".Oxigen_Too_high := FALSE;
       "Flag".STOP_HORN := TRUE;
   END_IF;
END_REGION

REGION Network 6: RO01 Oxigen low limit
   // no SCL statement known for SdCoil: written as a call
   #_w1 := "OFF" AND ("Manage_TC1_2".PID_Ref_Temp > 650.0) AND ("Data".Oxigen_RO01 <= 5);
   #_w2 := "OFF";
   SdCoil(in := #_w1, value := S5T#1M, operand := "Tag_106");
   IF #_w1 AND "Tag_106" THEN "Allarm".Oxigen_LOW := TRUE; END_IF;
   IF #_w2 AND "Flag".RESET_ALLARM AND "Allarm".Oxigen_LOW AND (("Data".Oxigen_RO01 >= 20) OR ("Manage_TC1_2".PID_Ref_Temp <= 650.0)) THEN
       "Allarm".Oxigen_LOW := FALSE;
   END_IF;
END_REGION

REGION Network 7: RO01-RO02 Signal compare FAULT
   // no SCL statement known for SdCoil: written as a call
   #_w1 := "ON" AND NOT "RO01-RO02control disable" AND ("Manage_TC1_2".PID_Ref_Temp > 650.0);
   IF #_w1 THEN #app01 := "Data".Oxigen_RO01 - "Data".Oxigen_RO02; END_IF;
   #_w2 := #_w1 AND ((#app01 < (-20)) OR (#app01 > 20));
   #_w3 := "ON";
   SdCoil(in := #_w2, value := S5T#1M, operand := "Tag_107");
   IF #_w2 AND "Tag_107" THEN "Allarm".RO01_Signal_Fault := TRUE; END_IF;
   IF #_w3 AND "Flag".RESET_ALLARM AND "Allarm".RO01_Signal_Fault THEN
       "Allarm".RO01_Signal_Fault := FALSE;
   END_IF;
END_REGION

REGION Network 8: TC01/TC02 signal compare fault
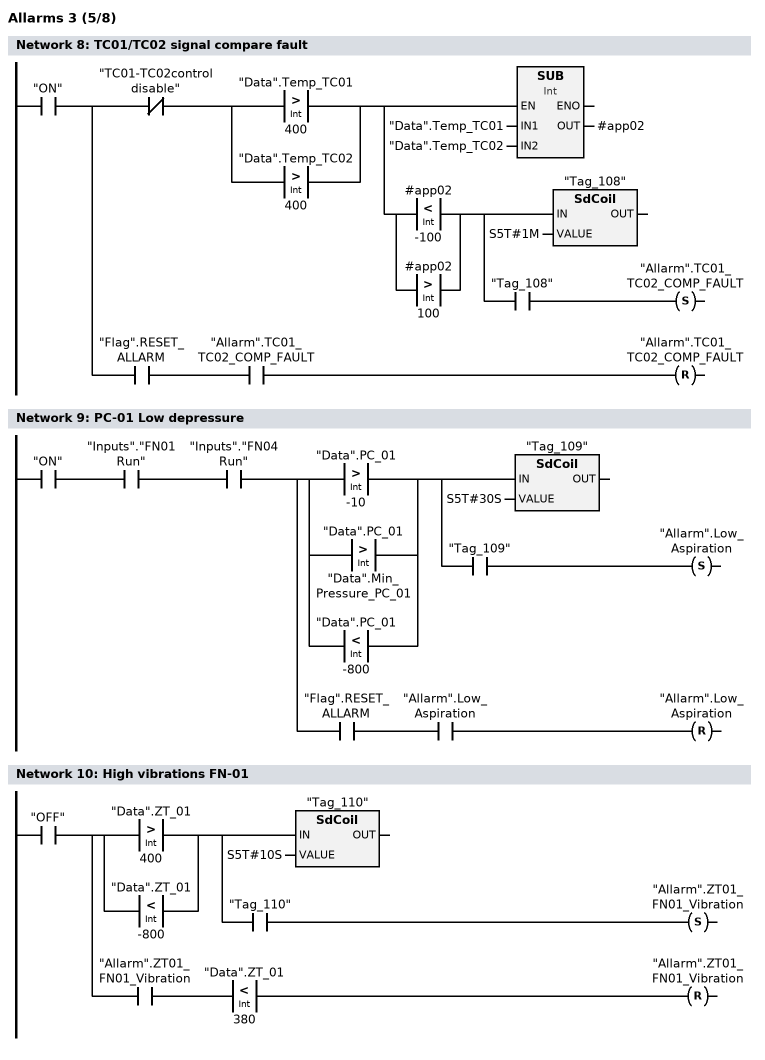
   // no SCL statement known for SdCoil: written as a call
   #_w1 := "ON" AND NOT "TC01-TC02control disable" AND (("Data".Temp_TC01 > 400) OR ("Data".Temp_TC02 > 400));
   IF #_w1 THEN #app02 := "Data".Temp_TC01 - "Data".Temp_TC02; END_IF;
   #_w2 := #_w1 AND ((#app02 < (-100)) OR (#app02 > 100));
   #_w3 := "ON";
   SdCoil(in := #_w2, value := S5T#1M, operand := "Tag_108");
   IF #_w2 AND "Tag_108" THEN "Allarm".TC01_TC02_COMP_FAULT := TRUE; END_IF;
   IF #_w3 AND "Flag".RESET_ALLARM AND "Allarm".TC01_TC02_COMP_FAULT THEN
       "Allarm".TC01_TC02_COMP_FAULT := FALSE;
   END_IF;
END_REGION

REGION Network 9: PC-01 Low depressure
   // no SCL statement known for SdCoil: written as a call
   #_w1 := "ON" AND "Inputs"."FN01 Run" AND "Inputs"."FN04 Run";
   #_w2 := #_w1 AND (("Data".PC_01 > (-10)) OR ("Data".PC_01 > "Data".Min_Pressure_PC_01) OR ("Data".PC_01 < (-800)));
   SdCoil(in := #_w2, value := S5T#30S, operand := "Tag_109");
   IF #_w2 AND "Tag_109" THEN "Allarm".Low_Aspiration := TRUE; END_IF;
   IF #_w1 AND "Flag".RESET_ALLARM AND "Allarm".Low_Aspiration THEN "Allarm".Low_Aspiration := FALSE; END_IF;
END_REGION

REGION Network 10: High vibrations FN-01
   // no SCL statement known for SdCoil: written as a call
   #_w1 := "OFF" AND (("Data".ZT_01 > 400) OR ("Data".ZT_01 < (-800)));
   #_w2 := "OFF";
   SdCoil(in := #_w1, value := S5T#10S, operand := "Tag_110");
   IF #_w1 AND "Tag_110" THEN "Allarm".ZT01_FN01_Vibration := TRUE; END_IF;
   IF #_w2 AND "Allarm".ZT01_FN01_Vibration AND ("Data".ZT_01 < 380) THEN
       "Allarm".ZT01_FN01_Vibration := FALSE;
   END_IF;
END_REGION

REGION Network 11: Max pressure PSH-02
